# B&R Automation Studio project perfxxl (part 4)

#### xml_interface.c
```c
#ifdef _DEFAULT_INCLUDES
	#include <AsDefault.h>
#endif
/***************************************************************************/
/*                                                                         */
/* Datei:    xml_interface.c                                               */
/*                                                                         */
/* Autor:    Herbert Aden, Krause-Biagosch GmbH                            */
/*                                                                         */
/* Abstrakt: Diese Task wartet darauf, daß sich ein TCP-IP Client am ein-  */
/*           gestellten Port anmeldet.   Wenn die Verbindung hergestellt   */
/*           worden ist, schickt der server zyklisch XML codierte          */
/*           wird versucht, die Verbindung wieder neu aufzubauen.          */
/*                                                                         */
/* Datum:    08.12.2006       letzte Änderungen: 25.01.2007  / HA          */
/*                                                                         */
/***************************************************************************/

/***** Include-Files: *****/
#include <Ethernet.h>
#include <string.h>
#include <ctype.h>
#include <visapi.h>
#include "asstring.h"
#include "glob_var.h"
#include "EGMglob_var.h"

/***** Variablen-/Konstantendeklaration: *****/
/* Anwendungsspezifische Konstanten: */
#define TCP_IP_PORT		2020				/* Port für Kommunikation */
#define SEND_BUFFER_LEN	3000				/* Buffer-Länge für das Senden */
#define RECV_BUFFER_LEN	150					/* Empfangs-Buffer Länge */
#define TIMEOUT			200					/* Abbruch nach TIMEOUT * Zykluszeit Sek.*/
#define	RCVTIMEOUT		200
#define MAXCLIENTS		5
#define	LIVEBYTECNT		160
#define SEND_EVERY_N_SEC 5					/* send every 5 seconds an xml message*/

/* sonstige Konstanten */
#define TCP_IP_OK			0
#define TCP_IP_NO_RCV_DATA	27211
#define TCP_IP_BUSY		65535
#define TCPIPMGR_TIMEOUT 14893
#define BUF_ZERO 14896

#define OPEN_PORT			0
#define WAIT_OPEN_PORT		1
#define SEND_DATA			2
#define WAIT_SEND_DATA		3
#define RECV_DATA			4
#define WAIT_RECV_DATA		5
#define CLOSE_PORT			6
#define WAIT_CLOSE_PORT		7

#define MAXERRORS			51

/* Strukturen fuer Ethernet-Libraray-Funktionen */
_LOCAL    TCPserv_typ         TCP_Server[MAXCLIENTS];
_LOCAL    TCPrecv_typ         TCP_Recv[MAXCLIENTS];
_LOCAL    TCPsend_typ         TCP_Send[MAXCLIENTS];
_LOCAL    TCPclose_typ        TCP_Close[MAXCLIENTS];

_LOCAL    SINT                Step[MAXCLIENTS];
_LOCAL    UINT                RcvLength;
_LOCAL    USINT               Count[MAXCLIENTS];
_LOCAL    USINT               SendDataCnt[MAXCLIENTS];
/* Buffer for XML Message */
_LOCAL    SINT                XMLBuffer[SEND_BUFFER_LEN];
_LOCAL    UINT                SendTimeout[MAXCLIENTS];
_LOCAL    UINT                Len;
_LOCAL    UINT                DataLock;

/* Variablen: */
static    SINT                SendBuffer[MAXCLIENTS][SEND_BUFFER_LEN];
static    SINT                RecvBuffer[MAXCLIENTS][RECV_BUFFER_LEN];
static    SINT                RecvData[MAXCLIENTS][RECV_BUFFER_LEN];
static    BOOL                CloseConnection[MAXCLIENTS];
static    int                 CurrentClient,parse;
static    int                 i;

static const char *ErrorTexts[] =
{
	"Not-Aus",
	"kein Antriebstakt",
	"Gummierung Füllstand zu niedrig",
	"Vorspülen Füllstand zu niedrig",
	"Nachspülen Füllstand zu niedrig",
	"Entwickler Füllstand zu niedrig",
	"Entwickler Temperatur zu niedrig",
	"Entwickler Temperatur zu hoch",
	"Nacherwärmung 1 Temperatur zu niedrig",
	"Nacherwärmung 1 Temperatur zu hoch",
	"Nacherwärmung 2 Temperatur zu niedrig",
	"Nacherwärmung 2 Temperatur zu hoch",
	"Plattenstau",
	"Entwickler zu alt",
	"E/A Modul nicht gefunden",
	"Nacherwärmung Temperatur-Sensor 1 defekt",
	"Nacherwärmung Temperatur-Sensor 2 defekt",
	"Nacherwärmung Umgebungs-Sensor defekt",
	"Entwickler Temperatur-Sensor defekt",
	"Nacherwärmung Heizung 1 defekt",
	"Nacherwärmung Heizung 2 defekt",
	"Vorspülstation: Befüllen fehlgeschlagen",
	"Nachspülstation: Befüllen fehlgeschlagen",
	"Entwickler Befüllen fehlgeschlagen",
	"Nacherwärmung 1 überhitzt",
	"Nacherwärmung 2 überhitzt",
	"Entwickler überhitzt",
	"Antrieb Geschwindigkeitsabweichung zu groß",
	"Temperatur Modul nicht gefunden",
	"Digitales Eingangsmodul nicht gefunden",
	"Digitales Ausgangsmodul nicht gefunden",
	"Analoges Ausgangsmodul nicht gefunden",
	"Versorgungsmodul nicht gefunden",
	"Gummierung: Kein Durchfluß",
	"Entwicklerzirkulation: Kein Durchfluß",
	"Vorspülen: Kein Durchfluß",
	"Nachspülen: Kein Durchfluß",
	"Regenerat Kanister leer",
	"Entwickler Kanister leer",
	"Nacherw.: Heizung 3 defekt",
	"Nacherw.: Heizung 4 defekt",
	"Nacherwärmung Kreis 3 Temp. zu niedrig",
	"Nacherwärmung Kreis 3 Temp. zu hoch",
	"Nacherwärmung Kreis 4 Temp. zu niedrig",
	"Nacherwärmung Kreis 4 Temp. zu hoch",
	"Nacherwärmung Kreis 3 überhitzt",
	"Nacherwärmung Kreis 4 überhitzt",
	"Nacherw.: Temperaturfühler 3 defekt",
	"Nacherw.: Temperaturfühler 4 defekt",
	"Abwassertank fast voll!",
	"Abwassertank voll, Maschine gestoppt!",
	"EOL",	/* End of Errorlist (for detection in loop) */
	" ",
	" ",
	" ",
	" ",
	" ",
	" ",
	" "
};

/***** INIT FUNKTION *******************************************************/
_INIT void init (void)
{
	int i;
	CurrentClient = 1;
	/* Initialisierung der TCP-IP Datenstrukturen: */

	for(i = 0;i<MAXCLIENTS;i++)
	{
		SendDataCnt[i] = 0;
		/* TCP-IP Client: */
		TCP_Server[i].enable	= TRUE;
		TCP_Server[i].porta	= TCP_IP_PORT+i;

		/* TCP-IP Client Senden: */
		TCP_Send[i].enable		= TRUE;
		TCP_Send[i].buffer		= (UDINT)&SendBuffer[i][0];
		TCP_Send[i].buflng		= SEND_BUFFER_LEN;

		/* TCP-IP Client Empfangen: */
		TCP_Recv[i].enable		= TRUE;
		TCP_Recv[i].buffer		= (UDINT)&RecvBuffer[i][0];
		TCP_Recv[i].mxbuflng	= RECV_BUFFER_LEN;

		/* TCP-IP Client schließen */
		TCP_Close[i].enable	= TRUE;

		Step[i] = OPEN_PORT;
		Count[i] = 0;
		CloseConnection[i] = 0;
	}

} /* Ende Funktion _INIT void init (void) */

void CreateXMLMessage( USINT *buf)
{
	char tmp[20];
	char TempError[64];
	int i,ErrorNumber;

	void AddVal2(USINT *buf, char *before,char *Value, char *after)
	{
		strcat(buf,before);
		strcat(buf,Value);
		strcat(buf,after);
	}

	strcpy(buf,"<KrauseMessage>\r\n\t<Bluefin>\r\n\t\t<MachineName>Bluefin</MachineName>\r\n");

			strcat(buf,"\t\t<MachineNumber>");
			strncat(buf,EGMGlobalParam.MachineNumber,9);
			strcat(buf,"</MachineNumber>\r\n");

			strcat(buf,"\t\t<MachineState>\r\n\t\t\t<State>");
/* Status Message*/
				strcpy(TempError,"No error");
				ErrorNumber = 0;
				switch (EGMState.mode)
				{
					case (M_OFF):
					case (M_CLEANING):
					case (M_INITCLEANING):
					{
					    if( !(ControlVoltageOk &&  ActivateControlVoltage) )
							strcat(buf,"EMERGENCY</State>\r\n\t\t\t<ErrorNumber>");
						else
							strcat(buf,"STANDBY</State>\r\n\t\t\t<ErrorNumber>");
						break;
					}
					case (M_AUTO):
					{
						switch (EGMState.state)
						{
							case (S_READY):
							{
								strcat(buf,"READY</State>\r\n\t\t\t<ErrorNumber>");
								break;
							}
							case (S_OFF):
							case (S_HEATING):
							{
								strcat(buf,"STANDBY</State>\r\n\t\t\t<ErrorNumber>");
								break;
							}
							case (S_STARTPROCESSING):
							case (S_PROCESSING):
							case (S_WAITFORSTANDBY):
							{
								strcat(buf,"BUSY</State>\r\n\t\t\t<ErrorNumber>");
								break;
							}
							case (S_ERROR):
							{
								BOOL Err = FALSE;
								strcat(buf,"ERROR</State>\r\n\t\t\t<ErrorNumber>");
/* find 1st error in list */
								for(i=0;i<MAXERRORS;i++)
								{
									if (EGM_AlarmBitField[i] == TRUE)
										break;
/* safety: detect End of Errorlist */
									if( strcmp(ErrorTexts[i],"EOL") == 0 )
									{
										Err = TRUE;
										break;
									}

								}
/* safety: End of Errorlist was detected */
								if(!Err && i<MAXERRORS)
								{
									strncpy(TempError,ErrorTexts[i],sizeof(TempError)-1);
									ErrorNumber = i;
								}
								else
								{
									ErrorNumber = 0;
								}
								break;
							}
						}
						break;
					}

				}
				itoa(ErrorNumber,(UDINT )&tmp[0]);
				strcat(buf,tmp);
				strcat(buf,"</ErrorNumber>\r\n\t\t\t<ErrorDescription>");
				strcat(buf,TempError);
				strcat(buf,"</ErrorDescription>\r\n\t\t\t<Errorlist>");
				for(i=0;i<EGM_MAXALARMS;i++)
				{
					if(EGM_AlarmBitField[i])
						strcat(buf,"1");
					else
						strcat(buf,"0");
				}

				strcat(buf,"</Errorlist>\r\n\t\t\t<StateCode>");
/* Emergency stop soll auch zu Error führen:*/
			    if( !(ControlVoltageOk &&  ActivateControlVoltage) )
					itoa(S_ERROR,(UDINT )&tmp[0]);
			    else
					itoa(EGMState.state,(UDINT )&tmp[0]);
				strcat(buf,tmp);
				strcat(buf,"</StateCode>\r\n\t\t</MachineState>\r\n\t\t<MachineParam>\r\n\t\t\t<PreHeat>\r\n");
/* Preheat values*/
					ftoa((REAL)EGMPreheat.RealTemp[0]/10.0,(UDINT )&tmp[0]);
					AddVal2(buf, "\t\t\t\t<Temperature1>\r\n\t\t\t\t\t<Description>Heating 1</Description>\r\n\t\t\t\t\t<Type>double</Type>\r\n\t\t\t\t\t<Value>", tmp,
					"</Value>\r\n\t\t\t\t\t<Unit>deg. C</Unit>\r\n\t\t\t\t</Temperature1>\r\n");
					ftoa((REAL)EGMPreheat.RealTemp[1]/10.0,(UDINT )&tmp[0]);
					AddVal2(buf, "\t\t\t\t<Temperature2>\r\n\t\t\t\t\t<Description>Heating 2</Description>\r\n\t\t\t\t\t<Type>double</Type>\r\n\t\t\t\t\t<Value>", tmp,
					"</Value>\r\n\t\t\t\t\t<Unit>deg. C</Unit>\r\n\t\t\t\t</Temperature2>\r\n");
					ftoa((REAL)EGMPreheat.RealTemp[2]/10.0,(UDINT )&tmp[0]);
					AddVal2(buf, "\t\t\t\t<Temperature3>\r\n\t\t\t\t\t<Description>Ambient</Description>\r\n\t\t\t\t\t<Type>double</Type>\r\n\t\t\t\t\t<Value>", tmp,
					"</Value>\r\n\t\t\t\t\t<Unit>deg. C</Unit>\r\n\t\t\t\t</Temperature3>\r\n\t\t\t</PreHeat>\r\n\t\t\t<Developer>\r\n");
/* Developer values */
					ftoa((REAL)EGMDeveloperTank.RealTemp/10.0,(UDINT )&tmp[0]);
					AddVal2(buf, "\t\t\t\t<Temperature1>\r\n\t\t\t\t\t<Description>Temperature of fluid</Description>\r\n\t\t\t\t\t<Type>double</Type>\r\n\t\t\t\t\t<Value>", tmp,
					"</Value>\r\n\t\t\t\t\t<Unit>deg. C</Unit>\r\n\t\t\t\t</Temperature1>\r\n");
					if(EGMDeveloperTank.LevelInRange)
						strcat(buf,"\t\t\t\t<LevelOK>\r\n\t\t\t\t\t<Description>Level of developer</Description>\r\n\t\t\t\t\t<Type>boolean</Type>\r\n\t\t\t\t\t<Value>true</Value>\r\n\t\t\t\t</LevelOK>\r\n\t\t\t</Developer>\r\n\t\t\t<Speeds>\r\n");
					else
						strcat(buf,"\t\t\t\t<LevelOK>\r\n\t\t\t\t\t<Description>Level of developer</Description>\r\n\t\t\t\t\t<Type>boolean</Type>\r\n\t\t\t\t\t<Value>false</Value>\r\n\t\t\t\t</LevelOK>\r\n\t\t\t</Developer>\r\n\t\t\t<Speeds>\r\n");
					ftoa(EGMGlobalParam.CurrentPlateSpeed,(UDINT )&tmp[0]);
					AddVal2(buf, "\t\t\t\t<PlateSpeedAct>\r\n\t\t\t\t\t<Description>Actual speed (measured)</Description>\r\n\t\t\t\t\t<Type>double</Type>\r\n\t\t\t\t\t<Value>", tmp,
					"</Value>\r\n\t\t\t\t\t<Unit>m per min</Unit>\r\n\t\t\t\t</PlateSpeedAct>\r\n");
					ftoa((EGMGlobalParam.MainMotorFactor*EGMMainMotor.RatedRpm),(UDINT )&tmp[0]);
					AddVal2(buf, "\t\t\t\t<PlateSpeedRef>\r\n\t\t\t\t\t<Description>Referenced speed</Description>\r\n\t\t\t\t\t<Type>double</Type>\r\n\t\t\t\t\t<Value>", tmp,
					"</Value>\r\n\t\t\t\t\t<Unit>m per min</Unit>\r\n\t\t\t\t</PlateSpeedRef>\r\n");
					itoa(EGMBrushMotor.RatedRpm*EGMGlobalParam.BrushFactor,(UDINT )&tmp[0]);
					AddVal2(buf, "\t\t\t\t<BrushSpeed>\r\n\t\t\t\t\t<Description>Speed of brushes</Description>\r\n\t\t\t\t\t<Type>int</Type>\r\n\t\t\t\t\t<Value>", tmp,
/*					"</Value>\r\n\t\t\t\t\t<Unit>rpm</Unit>\r\n\t\t\t\t</BrushSpeed>\r\n\t\t\t</Speeds>\r\n\t\t</MachineParam>\r\n\t</Bluefin>\r\n</KrauseMessage>\r\n");*/
/* *** */
					"</Value>\r\n\t\t\t\t\t<Unit>rpm</Unit>\r\n\t\t\t\t</BrushSpeed>\r\n\t\t\t</Speeds>\r\n\t\t</MachineParam>\r\n");
/* Verbrauchsdaten */
				strcat(buf,"\t\t<PlateCountValues>\r\n");
					itoa(OverallPlateCounter,(UDINT )&tmp[0]);
					AddVal2(buf, "\t\t\t<OverallPlates>\r\n\t\t\t\t<Description>Plates processed (overall)</Description>\r\n\t\t\t\t<Type>int</Type>\r\n\t\t\t\t<Value>", tmp,
					"</Value>\r\n\t\t\t\t<Unit>pcs.</Unit>\r\n\t\t\t</OverallPlates>\r\n");
					itoa(SessionPlateCounter,(UDINT )&tmp[0]);
					AddVal2(buf, "\t\t\t<SessionPlates>\r\n\t\t\t\t<Description>Plates processed since power on</Description>\r\n\t\t\t\t<Type>int</Type>\r\n\t\t\t\t<Value>", tmp,
					"</Value>\r\n\t\t\t\t<Unit>pcs.</Unit>\r\n\t\t\t</SessionPlates>\r\n");
					ftoa(OverallSqmCounter,(UDINT )&tmp[0]);
					AddVal2(buf, "\t\t\t<OverallSqm>\r\n\t\t\t\t<Description>Squaremeters processed (overall)</Description>\r\n\t\t\t\t<Type>double</Type>\r\n\t\t\t\t<Value>", tmp,
					"</Value>\r\n\t\t\t\t<Unit>sqm</Unit>\r\n\t\t\t</OverallSqm>\r\n");
					ftoa(SessionSqmCounter,(UDINT )&tmp[0]);
					AddVal2(buf, "\t\t\t<SessionSqm>\r\n\t\t\t\t<Description>Squaremeters processed since power on</Description>\r\n\t\t\t\t<Type>double</Type>\r\n\t\t\t\t<Value>", tmp,
					"</Value>\r\n\t\t\t\t<Unit>sqm</Unit>\r\n\t\t\t</SessionSqm>\r\n\t\t</PlateCountValues>\r\n");
/* Version */
				strcat(buf,"\t\t<Version>");
				strcat(buf,gVERSION);
				strcat(buf,"</Version>\r\n\t</Bluefin>\r\n</KrauseMessage>\r\n");

/* safety */
	if(strlen(buf) > SEND_BUFFER_LEN)
		buf[SEND_BUFFER_LEN-1] = 0;
	return;
}

/***** ZYKLISCHE FUNKTION **************************************************/
_CYCLIC void cyclic (void)
{

	if ( DataLock == 0 )
		CreateXMLMessage( (USINT *)&XMLBuffer[0] );

	for(CurrentClient = 0;CurrentClient<MAXCLIENTS;CurrentClient++)
	{
	/***** Öffnen des Ports ************************************************/
		if (Step[CurrentClient] == OPEN_PORT)
		{
 			CloseConnection[CurrentClient] = 0;
			/* 1. Aufruf der Funktion */
			TCPserv (&TCP_Server[CurrentClient]);
			/* Status prüfen: */
			if (TCP_Server[CurrentClient].status == TCP_IP_OK)
			{
				/* Port geöffnet */
				/* Identifier zuordnen ... */
				TCP_Send[CurrentClient].cident = TCP_Server[CurrentClient].cident;
				TCP_Recv[CurrentClient].cident = TCP_Server[CurrentClient].cident;
				TCP_Close[CurrentClient].cident = TCP_Server[CurrentClient].cident;
				/* ... und zum nächsten Schritt gehen */
				Step[CurrentClient] = RECV_DATA;
				SendTimeout[CurrentClient] = 0;
			}
		} /* if (Step == WAIT_OPEN_PORT) */

	/***** Daten Empfangen *************************************************/
		if (Step[CurrentClient] == RECV_DATA)
		{
			TCPrecv (&TCP_Recv[CurrentClient]);
			/* Status prüfen: */
			if (TCP_Recv[CurrentClient].status == TCP_IP_OK)
			{
				if(TCP_Recv[CurrentClient].rxbuflng == 0) /*CLOSE von Gegenstelle*/
				{
					Step[CurrentClient] = CLOSE_PORT;
					Count[CurrentClient] = 0;
				}
				else	/* Daten empfangen -> auswerten*/
				{
					parse = 0;
					/*einzelne Zeichen (via telnet)*/
					if(TCP_Recv[CurrentClient].rxbuflng < 3)
					{
						RecvData[CurrentClient][Count[CurrentClient]] = RecvBuffer[CurrentClient][0];
						Count[CurrentClient]++;
/* safety !*/
						if (Count[CurrentClient] >= RECV_BUFFER_LEN )
						{
							strcpy(SendBuffer[CurrentClient],"HEY! \a\aSTOP SENDING!!");
							Step[CurrentClient] = SEND_DATA;
							TCP_Send[CurrentClient].buffer		= (UDINT)&SendBuffer[CurrentClient];
							TCP_Send[CurrentClient].buflng = strlen(SendBuffer[CurrentClient]);
							Count[CurrentClient] = 0;
							parse = 0;
						}
						else
						if( RecvBuffer[CurrentClient][0] == 10 || RecvBuffer[CurrentClient][0] == 13 )
						{
							RecvData[CurrentClient][Count[CurrentClient]] = 0;
							parse = 1;
						}
					}
					else
					{
						memcpy(RecvData[CurrentClient],RecvBuffer[CurrentClient],TCP_Recv[CurrentClient].rxbuflng);
						Count[CurrentClient] = TCP_Recv[CurrentClient].rxbuflng;
						parse = 1;
					}

					if(parse)
					{
						i=0;
						while(  ( RecvData[CurrentClient][i] != 0 )
						     && ( i < RECV_BUFFER_LEN) )
						{
							RecvData[CurrentClient][i] = toupper( RecvData[CurrentClient][i] );
							i++;
						}
						RecvData[CurrentClient][Count[CurrentClient]-1] = 0;

						if (strncmp(RecvData[CurrentClient],"BYE",3) == 0
						||	strncmp(RecvData[CurrentClient],"QUIT",4) == 0
						||	strncmp(RecvData[CurrentClient],"EXIT",4) == 0)
						{
							strcpy(SendBuffer[CurrentClient],"Good bye, cu next time...\r\n");
							CloseConnection[CurrentClient] = 1;
						}
						Step[CurrentClient] = SEND_DATA;
						TCP_Send[CurrentClient].buffer		= (UDINT)&SendBuffer[CurrentClient];
						TCP_Send[CurrentClient].buflng = strlen(SendBuffer[CurrentClient]);
						Count[CurrentClient] = 0;
						parse = 0;
					}
					SendDataCnt[CurrentClient]=0;
				}
			}
			else
			{
/*nothing received: ok, send from time to time*/
				SendDataCnt[CurrentClient]++;
				if( SendDataCnt[CurrentClient] >= 10*SEND_EVERY_N_SEC)
				{
					memcpy(SendBuffer[CurrentClient],XMLBuffer,sizeof(XMLBuffer));
					TCP_Send[CurrentClient].buflng = strlen(SendBuffer[CurrentClient]);
					Step[CurrentClient] = SEND_DATA;
					SendDataCnt[CurrentClient] = 0;
				}
			}
		}

/************** senden ****************************/

		if (Step[CurrentClient] == SEND_DATA)
		{

			TCPsend (&TCP_Send[CurrentClient]);
			/* Status prüfen: */
			if (TCP_Send[CurrentClient].status == TCP_IP_OK)
			{
				/* Senden war OK */
				if (CloseConnection[CurrentClient])
					Step[CurrentClient] = CLOSE_PORT;
				else
					Step[CurrentClient] = RECV_DATA;
				CloseConnection[CurrentClient] = 0;
				SendTimeout[CurrentClient] = 0;
			}
			else
			if (TCP_Send[CurrentClient].status == TCP_IP_BUSY)
			{
			/* VOID, just wait*/
			}
			else
			if (TCP_Send[CurrentClient].status == ERR_ETH_NET_SLOW)
			{
			/* Check for timeout, after 3 sec close the port and wait for reconnection */
				SendTimeout[CurrentClient]++;
				if(SendTimeout[CurrentClient] > 30) /* 3 sec*/
					Step[CurrentClient] = CLOSE_PORT;
			}
			else
			if (TCP_Send[CurrentClient].status == TCPIPMGR_TIMEOUT)
			{
			/* VOID, just wait*/
			}
			else	/* any other state, close after a certain time*/
			{
				SendTimeout[CurrentClient]++;
				if(SendTimeout[CurrentClient] > 30) /* 3 sec*/
					Step[CurrentClient] = CLOSE_PORT;
			}
		}

	/***** Port schließen **************************************************/
		if (Step[CurrentClient] == CLOSE_PORT)
		{
			SendTimeout[CurrentClient] = 0;
			TCPclose (&TCP_Close[CurrentClient]);
			/* Status prüfen: */
			if (TCP_Close[CurrentClient].status == TCP_IP_OK)
			{
				/* Port geschlossen, neu öffnen: */
				Step[CurrentClient] = OPEN_PORT;
			}
		} /* if (Step == WAIT_CLOSE_PORT) */

	} /*for*/

} /* Ende Funktion _CYCLIC void cyclic (void) */

/* ENDE */
```

### Program Logical/bluefin (ANSIC, version 0.00.0)

#### ifbluefin.c
```c
#ifdef _DEFAULT_INCLUDES
	#include <AsDefault.h>
#endif
/*
                             *******************
******************************* C SOURCE FILE *******************************
**                           *******************                           **
**                                                                         **
** project  : LS JET II                                                    **
** filename : IFBLUEFIN.C                                                  **
** version  : 1.01                                                         **
** date     : 23.06.2010                                                   **
**                                                                         **
*****************************************************************************
** Abstract                                                                **
** ========                                                                **
** -Interface to Bluefin via CAN using the IMA library                     **
**  Needs Dataobject DO_IMA                                                **
** -TCPIP Server for data transfer to BluefinServer, takes messages        **
**  from Bluefin (in connected XMLBuffer array) and transfers this         **
**  to all connected clients (max 3) periodically                          **
**  if no connection to Bluefin is established the message "BLUEFIN OFF"   **
**  is sent periodically                                                   **
**                                                                         **
** Copyright (c) 2006, Krause-Biagosch GmbH                                **
** All rights reserved.                                                    **
**                                                                         **
*****************************************************************************
VERSION HISTORY:
----------------
Version     : 1.00
Date        : 15.01.2007
Revised by  : Herbert Aden
Description : Original version.

Version     : 1.01
Date        : 23.06.2010
Revised by  : Herbert Aden
Description : Improved version from LSJet.

*/
#define _IFBLUEFIN_C_SRC

/****************************************************************************/
/**                                                                        **/
/**                           INCLUDE FILES                                **/
/**                                                                        **/
/****************************************************************************/
#include "glob_var.h"
#include "egmglob_var.h"
#include "in_out.h"
#include <AsIMA.h>
#include <Ethernet.h>
#include <string.h>
#include <ctype.h>
#include "asstring.h"

/****************************************************************************/
/**                                                                        **/
/**                       DEFINITIONS AND MACROS                           **/
/**                                                                        **/
/****************************************************************************/
#define IMA_CONN_OK          (0)

#define TCP_IP_PORT		2020				/* Port für Kommunikation */
#define SEND_BUFFER_LEN	3000				/* Buffer-Länge für das Senden */
#define OLD_SEND_BUFFER_LEN	2500				/* XML Buffer-Länge für Bluefin <=2.10*/
#define RECV_BUFFER_LEN	150					/* Empfangs-Buffer Länge */
#define TIMEOUT			200					/* Abbruch nach TIMEOUT * Zykluszeit Sek.*/
#define	RCVTIMEOUT		200
#define MAXCLIENTS		3
#define	LIVEBYTECNT		160
#define SEND_EVERY_N_SEC 3					/* send every 5 seconds an xml message*/

/* sonstige Konstanten */
#define TCP_IP_OK			0
#define TCP_IP_NO_RCV_DATA	27211
#define TCP_IP_BUSY		65535
#define TCPIPMGR_TIMEOUT 14893
#define BUF_ZERO 14896

#define OPEN_PORT			0
#define WAIT_OPEN_PORT		1
#define SEND_DATA			2
#define WAIT_SEND_DATA		3
#define RECV_DATA			4
#define WAIT_RECV_DATA		5
#define CLOSE_PORT			6
#define WAIT_CLOSE_PORT		7
#define WAIT				8
#define PREPARE_SEND_DATA   9

/****************************************************************************/
/**                                                                        **/
/**                      TYPEDEFS AND STRUCTURES                           **/
/**                                                                        **/
/****************************************************************************/
/* NONE */

/****************************************************************************/
/**                                                                        **/
/**                      PROTOTYPES OF LOCAL FUNCTIONS                     **/
/**                                                                        **/
/****************************************************************************/
/* NONE */

/****************************************************************************/
/**                                                                        **/
/**                      EXPORTED VARIABLES                                **/
/**                                                                        **/
/****************************************************************************/
/* NONE */

/****************************************************************************/
/**                                                                        **/
/**                           GLOBAL VARIABLES                             **/
/**                                                                        **/
/****************************************************************************/

/****************************************************************************/
/**                                                                        **/
/**                      TASK-LOCAL VARIABLES                              **/
/**                                                                        **/
/****************************************************************************/
_LOCAL    INT                 IMAStatusInit,IMAStatusComm;
_LOCAL    imaInfoStruct       errorInfo,ConnInfoPV,ConnInfoAUX;
_LOCAL    UDINT               IMAident;

_LOCAL    INT                 IMAStatusInitVCP,IMAStatusInitXSOld,IMAStatusCommVCP,IMAStatusCommXSOld;
_LOCAL    imaInfoStruct       errorInfoVCP,ConnInfoPVVCP,ConnInfoAUXVCP;
_LOCAL    imaInfoStruct       errorInfoXSOld,ConnInfoPVXSOld,ConnInfoAUXXSOld;
_LOCAL    UDINT               IMAidentVCP,IMAidentXSOld;

_LOCAL    UINT                byte_link_cnt;

/* structs for Ethernet-Library-Functions */
_LOCAL	TCPserv_typ			TCP_Server[MAXCLIENTS];
_LOCAL	TCPrecv_typ			TCP_Recv[MAXCLIENTS];
_LOCAL	TCPsend_typ			TCP_Send[MAXCLIENTS];
_LOCAL	TCPclose_typ		TCP_Close[MAXCLIENTS];
_LOCAL	SINT	Step[MAXCLIENTS];
_LOCAL	UINT	SendTimeout[MAXCLIENTS];
_LOCAL	UINT	RcvLength;

/* Buffer for XML Message */
_LOCAL SINT	XMLBuffer[SEND_BUFFER_LEN];
_LOCAL SINT	OldXMLBuffer[OLD_SEND_BUFFER_LEN];
_LOCAL UINT EnablePVComm;
_LOCAL UINT	DataLock;
_LOCAL BOOL                CAN_EGM1;
_LOCAL BOOL                CAN_EGM2;
_LOCAL BOOL                CAN_VCP;
_LOCAL STRING              BFVERSION[9];
_LOCAL UINT                IMACommStep;
_LOCAL UINT                VisConnOK;

/****************************************************************************/
/**                                                                        **/
/**                    MODULE-LOCAL VARIABLES                              **/
/**                                                                        **/
/****************************************************************************/
/* for IMA Comm */
static    STRING              DOName[32]="do_ima";
static    STRING              DONameVCP[32]="do_vcp";
static    STRING              DONameXSOld[32]="do_xsold";
/* for Ethernet server */
static    SINT                SendBuffer[MAXCLIENTS][SEND_BUFFER_LEN];
static    SINT                RecvBuffer[MAXCLIENTS][RECV_BUFFER_LEN];
static    SINT                RecvData[MAXCLIENTS][RECV_BUFFER_LEN];

static    int                 CurrentClient,parse;
static    USINT               Count[MAXCLIENTS];
static    int                 i;
static    USINT               SendDataCnt[MAXCLIENTS];
static    BOOL                CloseConnection[MAXCLIENTS];
static    UINT                NumberOfFreePorts;
static    UINT                WaitCounter[MAXCLIENTS];
static    BOOL                ConnectedTo3000Byte;
/****************************************************************************/
/**                                                                        **/
/**                          LOCAL FUNCTIONS                               **/
/**                                                                        **/
/****************************************************************************/
_INIT void InitFunc(void)
{
#ifdef MODE_PERFORMANCE
	int i;
	ConnectedTo3000Byte = FALSE;
	IMACommStep = 0;
	IMAStatusInit = IMAinit((UDINT)DOName, &errorInfo, &IMAident);
	IMAStatusInitVCP = IMAinit((UDINT)DONameVCP, &errorInfoVCP, &IMAidentVCP);
	IMAStatusInitXSOld = IMAinit((UDINT)DONameXSOld, &errorInfoXSOld, &IMAidentXSOld);

	CurrentClient = 1;
	/* Initialise TCP-IP Data structs: */
	for(i = 0;i<MAXCLIENTS;i++)
	{
		SendDataCnt[i] = 0;
		/* TCP-IP Client: */
		TCP_Server[i].enable	= TRUE;
		TCP_Server[i].porta	= TCP_IP_PORT+i;

		/* TCP-IP Client Senden: */
		TCP_Send[i].enable		= TRUE;
		TCP_Send[i].buffer		= (UDINT)&SendBuffer[i][0];
		TCP_Send[i].buflng		= SEND_BUFFER_LEN;

		/* TCP-IP Client Empfangen: */
		TCP_Recv[i].enable		= TRUE;
		TCP_Recv[i].buffer		= (UDINT)&RecvBuffer[i][0];
		TCP_Recv[i].mxbuflng	= RECV_BUFFER_LEN;

		/* TCP-IP Client schließen */
		TCP_Close[i].enable	= TRUE;

		Step[i] = OPEN_PORT;
		Count[i] = 0;
		CloseConnection[i] = 0;
	}
	NumberOfFreePorts = MAXCLIENTS;
	AlarmBitField[35] = FALSE;
	VisConnOK = 0;
#endif
}

_CYCLIC void CyclicFunc(void)
{
/*****************************************************************************/
/* get data from Bluefin via INA comm */
/*****************************************************************************/

#ifdef MODE_BOTH
/* Performance und Bluefin: EGM Signale direkt aus der Software*/
	StatusEGM1 = NoError;
	StatusEGM2 = Ready;
	VCP = VCP_OK;
#else
/* Performance allein: EGM Signale via CAN Anbindung oder Eingänge*/

	if(IMAStatusInit == IMA_OK)  /* Init was OK (should always be the case) */
	{
		switch (IMACommStep)
		{
			case 0:
			{ /* Versuch, mit der neuesten Version zu connecten */
				IMAStatusCommVCP = IMAcomm(IMAidentVCP, &ConnInfoPVVCP, &ConnInfoAUXVCP);

				if(IMAStatusCommVCP == IMA_OK)
				{
/*
 * Bluefin XS Version bis 3.04 hat 2500 Byte Puffer, deswegen dann anderen
 * Verbindungs DB benutzen
 */
					if(  (BFVERSION[0] == '3')
					  && (BFVERSION[2] == '0')
					  && (BFVERSION[5] != 'L') /* LC Version erkennen, die hat nämlich
					                            * auch 3000 Byte und VCP Verbindung
					                            */
				  )
					{
						IMACommStep = 20;
					}
					else
					{
						ConnectedTo3000Byte = TRUE;
						StatusEGM1 = CAN_EGM1;
						StatusEGM2 = CAN_EGM2;
						VCP = CAN_VCP;
						AlarmBitField[35] = FALSE;
						VisConnOK = 1;

						if(NumberOfFreePorts < MAXCLIENTS)
							EnablePVComm = 1;
						else
							EnablePVComm = 0;
					}
				}
				else /* fehlgeschlagen: Verbindung beenden und alte Version probieren */
					IMACommStep = 20;
				break;
			}

			case 20:
			{ /* Versuch, mit Version XS mit 2500 Byte zu connecten */
				IMAStatusCommXSOld = IMAcomm(IMAidentXSOld, &ConnInfoPVXSOld, &ConnInfoAUXXSOld);

				if(IMAStatusCommXSOld == IMA_OK)
				{
					ConnectedTo3000Byte = FALSE;
					StatusEGM1 = CAN_EGM1;
					StatusEGM2 = CAN_EGM2;
					VCP = CAN_VCP;
					AlarmBitField[35] = FALSE;
					VisConnOK = 1;

					if(NumberOfFreePorts < MAXCLIENTS)
						EnablePVComm = 1;
					else
						EnablePVComm = 0;
				}
				else /* fehlgeschlagen: Verbindung beenden und alte Version probieren */
					IMACommStep = 30;
				break;
			}

			case 30:
			{ /* Versuch, mit der alten Version zu connecten */
				IMAStatusComm = IMAcomm(IMAident, &ConnInfoPV, &ConnInfoAUX);

				if(IMAStatusComm == IMA_OK)
				{
/*
 * Bluefin XS Version bis 3.04 hat auch 2500 Byte Puffer, wird nicht per Fehler erkannt,
 * weil hier (im hierzu gehörigen DB) nicht auf CAN_VCP zugegriffen wird
 * deshalb über Versionsnummer
 */
					if(  (BFVERSION[0] == '3')
					  )
					{
						IMACommStep = 20;
					}
					else
					{
						ConnectedTo3000Byte = FALSE;
						StatusEGM1 = CAN_EGM1;
						StatusEGM2 = CAN_EGM2;
						VCP = CAN_VCP;
						AlarmBitField[35] = FALSE;
						VisConnOK = 1;

						if(NumberOfFreePorts < MAXCLIENTS)
							EnablePVComm = 1;
						else
							EnablePVComm = 0;
					}
				}
				else /* fehlgeschlagen: Fehlermeldung und von vorn beginnen */
				{
					ConnInfoPVVCP.commandClearError = TRUE;
					ConnInfoPVXSOld.commandClearError = TRUE;
					ConnInfoPV.commandClearError = TRUE;
					VisConnOK = 0;
					IMACommStep = 0;
					StatusEGM1 = InEGM1;
					StatusEGM2 = InEGM2;
					VCP = In_VCPOK;
					break;
				}
				break;
			}
		}/*switch*/
	}
	else  /* comm not OK: EGM signals via Digital inputs*/
	{
		ConnectedTo3000Byte = FALSE;
		StatusEGM1 = InEGM1;
		StatusEGM2 = InEGM2;
		VCP = In_VCPOK;
	}

/*****************************************************************************/
/* TCP/IP Server */
/*****************************************************************************/
	NumberOfFreePorts = 0;

	for(CurrentClient = 0;CurrentClient<MAXCLIENTS;CurrentClient++)
	{
	/***** Öffnen des Ports ************************************************/
		if (Step[CurrentClient] == OPEN_PORT)
		{
 			CloseConnection[CurrentClient] = 0;
			/* 1. Aufruf der Funktion */
			TCPserv (&TCP_Server[CurrentClient]);
			/* Status prüfen: */
			if (TCP_Server[CurrentClient].status == TCP_IP_OK)
			{
				/* Port geöffnet */
				/* Identifier zuordnen ... */
				TCP_Send[CurrentClient].cident = TCP_Server[CurrentClient].cident;
				TCP_Recv[CurrentClient].cident = TCP_Server[CurrentClient].cident;
				TCP_Close[CurrentClient].cident = TCP_Server[CurrentClient].cident;
				/* ... und zum nächsten Schritt gehen */
				Step[CurrentClient] = RECV_DATA;
				SendTimeout[CurrentClient] = 0;
			}
			else
				NumberOfFreePorts++;
		} /* if (Step == WAIT_OPEN_PORT) */

	/***** Daten Empfangen *************************************************/
		if (Step[CurrentClient] == RECV_DATA)
		{
			TCPrecv (&TCP_Recv[CurrentClient]);
			/* Status prüfen: */
			if (TCP_Recv[CurrentClient].status == TCP_IP_OK)
			{
				if(TCP_Recv[CurrentClient].rxbuflng == 0) /*CLOSE von Gegenstelle*/
				{
					Step[CurrentClient] = CLOSE_PORT;
					Count[CurrentClient] = 0;
				}
				else	/* Daten empfangen -> auswerten*/
				{
					parse = 0;
					/*einzelne Zeichen (via telnet)*/
					if(TCP_Recv[CurrentClient].rxbuflng < 3)
					{
						RecvData[CurrentClient][Count[CurrentClient]] = RecvBuffer[CurrentClient][0];
						Count[CurrentClient]++;
/* safety !*/
						if (Count[CurrentClient] >= RECV_BUFFER_LEN )
						{
							strcpy(SendBuffer[CurrentClient],"HEY! \a\aSTOP SENDING!!");
							Step[CurrentClient] = SEND_DATA;
							TCP_Send[CurrentClient].buffer		= (UDINT)&SendBuffer[CurrentClient];
							TCP_Send[CurrentClient].buflng = strlen(SendBuffer[CurrentClient]);
							Count[CurrentClient] = 0;
							parse = 0;
						}
						else
						if( RecvBuffer[CurrentClient][0] == 10 || RecvBuffer[CurrentClient][0] == 13 )
						{
							RecvData[CurrentClient][Count[CurrentClient]] = 0;
							parse = 1;
						}
					}
					else
					{
						memcpy(RecvData[CurrentClient],RecvBuffer[CurrentClient],TCP_Recv[CurrentClient].rxbuflng);
						Count[CurrentClient] = TCP_Recv[CurrentClient].rxbuflng;
						parse = 1;
					}

					if(parse)
					{
						i=0;
						while(  ( RecvData[CurrentClient][i] != 0 )
						     && ( i < RECV_BUFFER_LEN) )
						{
							RecvData[CurrentClient][i] = toupper( RecvData[CurrentClient][i] );
							i++;
						}
						RecvData[CurrentClient][Count[CurrentClient]-1] = 0;

						if (strncmp(RecvData[CurrentClient],"BYE",3) == 0
						||	strncmp(RecvData[CurrentClient],"QUIT",4) == 0
						||	strncmp(RecvData[CurrentClient],"EXIT",4) == 0)
						{
							strcpy(SendBuffer[CurrentClient],"Good bye, cu next time...\r\n");
							CloseConnection[CurrentClient] = 1;
						}
						Step[CurrentClient] = SEND_DATA;
						TCP_Send[CurrentClient].buffer		= (UDINT)&SendBuffer[CurrentClient];
						TCP_Send[CurrentClient].buflng = strlen(SendBuffer[CurrentClient]);
						Count[CurrentClient] = 0;
						parse = 0;
					}
					SendDataCnt[CurrentClient]=0;
				}
			}
			else
			{
/*nothing received: ok, send from time to time*/
				SendDataCnt[CurrentClient]++;
				if( SendDataCnt[CurrentClient] >= 10*SEND_EVERY_N_SEC )
				{
					if(  (IMAStatusComm    == IMA_OK)
					 ||  (IMAStatusCommVCP == IMA_OK)
					 ||  (IMAStatusCommXSOld == IMA_OK) )
					{
						DataLock = 1;
						Step[CurrentClient] = WAIT;
						SendDataCnt[CurrentClient] = 0;
						WaitCounter[CurrentClient] = 0;
					}
					else
					{
						strcpy(SendBuffer[CurrentClient],"BLUEFIN OFF");
						TCP_Send[CurrentClient].buflng = strlen(SendBuffer[CurrentClient]);
						Step[CurrentClient] = SEND_DATA;
						SendDataCnt[CurrentClient] = 0;
					}
				}
			}
		}

/* SENDEDATEN VORBEREITEN */
		if (Step[CurrentClient] == PREPARE_SEND_DATA)
		{
			if(ConnectedTo3000Byte)
			{
/* Bluefin XS Version mit 3000 Byte xml Puffer */
				if( strncmp(XMLBuffer,"<KrauseMessage>",15) == 0 )
				{
					memcpy(SendBuffer[CurrentClient],XMLBuffer,sizeof(XMLBuffer));
					TCP_Send[CurrentClient].buflng = strlen(SendBuffer[CurrentClient]);
					Step[CurrentClient] = SEND_DATA;
					SendDataCnt[CurrentClient] = 0;
					DataLock = 0;
				}
			}
			else
			{
/* Bluefin standard Version mit 2500 Byte xml Puffer */
				if( strncmp(OldXMLBuffer,"<KrauseMessage>",15) == 0 )
				{
					memcpy(SendBuffer[CurrentClient],OldXMLBuffer,sizeof(OldXMLBuffer));
					SendBuffer[CurrentClient][sizeof(OldXMLBuffer)-1] = 0;
					TCP_Send[CurrentClient].buflng = strlen(SendBuffer[CurrentClient]);
					Step[CurrentClient] = SEND_DATA;
					SendDataCnt[CurrentClient] = 0;
					DataLock = 0;
				}
			}
		}

/************** senden ****************************/

		if (Step[CurrentClient] == SEND_DATA)
		{

			TCPsend (&TCP_Send[CurrentClient]);
			/* Status prüfen: */
			if (TCP_Send[CurrentClient].status == TCP_IP_OK)
			{
				/* Senden war OK */
				if (CloseConnection[CurrentClient])
					Step[CurrentClient] = CLOSE_PORT;
				else
					Step[CurrentClient] = RECV_DATA;
				CloseConnection[CurrentClient] = 0;
				SendTimeout[CurrentClient] = 0;
			}
			else
			if (TCP_Send[CurrentClient].status == TCP_IP_BUSY)
			{
			/* VOID, just wait*/
			}
			else
			if (TCP_Send[CurrentClient].status == ERR_ETH_NET_SLOW)
			{
			/* Check for timeout, after 3 sec close the port and wait for reconnection */
				SendTimeout[CurrentClient]++;
				if(SendTimeout[CurrentClient] > 30) /* 3 sec*/
					Step[CurrentClient] = CLOSE_PORT;
			}
			else
			if (TCP_Send[CurrentClient].status == TCPIPMGR_TIMEOUT)
			{
			/* VOID, just wait*/
			}
			else	/* any other state, close after a certain time*/
			{
				SendTimeout[CurrentClient]++;
				if(SendTimeout[CurrentClient] > 30) /* 3 sec*/
					Step[CurrentClient] = CLOSE_PORT;
			}
		}

	/***** Port schließen **************************************************/
		if (Step[CurrentClient] == CLOSE_PORT)
		{
			SendTimeout[CurrentClient] = 0;
			TCPclose (&TCP_Close[CurrentClient]);
			/* Status prüfen: */
			if (TCP_Close[CurrentClient].status == TCP_IP_OK)
			{
				/* Port geschlossen, neu öffnen: */
				Step[CurrentClient] = OPEN_PORT;
			}
		} /* if (Step == WAIT_CLOSE_PORT) */

		if (Step[CurrentClient] == WAIT)
		{
			WaitCounter[CurrentClient]++;
			if( WaitCounter[CurrentClient] > 20 )
			{
				Step[CurrentClient] = PREPARE_SEND_DATA;
				WaitCounter[CurrentClient] = 0;
			}
		} /* if (Step == WAIT) */

	} /*for*/
#endif

}
```

### Program Logical/hwconfig (ANSIC, version 0.00.0)

#### hwconfig.c
```c
#ifdef _DEFAULT_INCLUDES
	#include <AsDefault.h>
#endif
/* ===================================================== HEADER FILES ===================================================== */

#include <bur/plc.h>
#include <bur/plctypes.h>
#include <sys_lib.h>
#include <asiomman.h>
#include <brsystem.h>
#include <standard.h>
#include "auxfunc.h"

/* ===================================================== VARAIBLE DECLARATION ==================================================== */

#define ERR_FUB_BUSY 65535
#define MAXHWMODULES (20)
#define ERR_IO_CHECK_NOMODULE (5555)

typedef struct
{
	STRING Name[20];
	UINT HWStatus;
	USINT HWFamily;
	USINT HWUseType;
	USINT HWModuleTyp;
	USINT HWMasterNo;
	USINT HWSlaveNo;
	USINT HWModuleAdr;
	USINT HWSlotNo;
}HW_Info_typ;

_GLOBAL UINT        change_config;                  /* indicates if configuration should be changed */
_GLOBAL UINT        config;                         /* indicates if configuration should be changed */
_GLOBAL USINT       step;                           /* step for the main routine */
_LOCAL  USINT       status_message[128];            /* shows the status of the program */

/* CYCLIC */
_LOCAL  AsIOMMCreate_typ    AsIOMMCreate_Mod;       /* function for creating the new BR module on the target */
_LOCAL  AsIOMMRemove_typ    AsIOMMRemove_Mod;       /* function for removing the BR module on the target */
_LOCAL  AsIOMMCopy_typ      AsIOMMCopy_Mod;         /* function for copying the BR module to a datamodule */
_LOCAL  USINT           error_string[128];

/* shows the last error which occured */
_LOCAL  USINT           error_step;                 /* step where the error occurred */
_LOCAL  UINT            error_status;               /* status of the FBK where the error occured */
_LOCAL  BOOL            error;                      /* shows if an error occurred */
static TON_10ms_typ     WaitTimer;                  /*waits before actually changing config*/
/************************************/

_LOCAL	HWInfo_typ HWInfo_01;

_LOCAL  BOOL            CopyArConfig,CopyIomap,InstallConfig1,InstallConfig2;
_LOCAL  BOOL            next;
_LOCAL	HW_Info_typ		myHWInfo[MAXHWMODULES];
_LOCAL	INT				cnt;
_GLOBAL SINT            IOConfiguration _VAR_RETAIN,NewIOConfig	_VAR_RETAIN;
_GLOBAL SINT 			IOChangeStep	_VAR_RETAIN;

_INIT void InitialisierungsProgramm(void) {
        HWInfo_01.enable = 1;     /* Funktionsblock wird nur ausgeführt
                                   wenn ENABLE <> 0 ist. */
        HWInfo_01.first = 1;      /* Bestimmen des Hardwaremoduls auf dem die
                                   Funktion angewendet werden soll. */
        cnt = 0;
        next = 1;

        InstallConfig1 = 0;
        InstallConfig2 = 0;
        NewIOConfig = 0;
		WaitTimer.IN = 0;
}

_CYCLIC void cyclic( void )
{
	if(next || HWInfo_01.first)
	{
        HWInfo_01.pName = (UDINT) &(myHWInfo[cnt].Name);
        HWInfo(&HWInfo_01);
        myHWInfo[cnt].HWStatus    = HWInfo_01.status;     /* Fehlernummer, 0 ist kein Fehler. */
        myHWInfo[cnt].HWFamily    = HWInfo_01.family;     /* Familienbezeichnung */
        myHWInfo[cnt].HWUseType   = HWInfo_01.usetype;   /* Hardware-Typ */
        myHWInfo[cnt].HWModuleTyp = HWInfo_01.module_typ; /* Typcode des Moduls */
        myHWInfo[cnt].HWMasterNo  = HWInfo_01.master_no;   /* Logische Nummer des IO-Masters, des RIO-Masters bzw.
                                                des CAN-Busses bei CANIO. */
        myHWInfo[cnt].HWSlaveNo   = HWInfo_01.slave_no;     /* Slave Nummer */
        myHWInfo[cnt].HWModuleAdr = HWInfo_01.module_adr;    /* Moduladresse des Hardwaremoduls */
        myHWInfo[cnt].HWSlotNo    = HWInfo_01.slot_no;          /* Steckplatz des Einschub-oder Anpassungsmoduls */

		HWInfo_01.first = 0;
		if(cnt < MAXHWMODULES)
			cnt++;

		if( (HWInfo_01.status == ERR_IO_CHECK_NOMODULE)
		 || (cnt >= MAXHWMODULES)
		  )
		{
			next = 0;
			cnt = 0;
		}
	}

/***********************************************************/

/* change request from pics task (user changes config.)*/

	if(NewIOConfig == 1)
	{
		InstallConfig1 = 1;
		NewIOConfig = 0;
	}
	else
	if(NewIOConfig == 2)
	{
		InstallConfig2 = 1;
		NewIOConfig = 0;
	}

	TON_10ms(&WaitTimer);

	switch (step)
	{
		case 0:
		{
            if(IOChangeStep != 0)
            {
	            if(IOChangeStep == 12)
	            	InstallConfig1 = 1;
	            if(IOChangeStep == 13)
	            	InstallConfig2 = 1;
            	step = 20;
            	IOChangeStep = 0;
            	break;
            }

			if(CopyArConfig)
			{
				CopyArConfig = 0;
				step = 1;
				break;
			}
			if(CopyIomap)
			{
				CopyIomap = 0;
				step = 2;
				break;
			}

			if(InstallConfig1 || InstallConfig2)
			{
				if(WaitTimer.Q)
				{
					WaitTimer.IN = 0;
					step = 5;
					break;
				}
				WaitTimer.IN = 1;
				WaitTimer.PT = 200;
				ShowMessage(128,129,0,INFO,NONE, 1);
				break;
			}
			break;
		}
		case 1:
		{
            AsIOMMCopy_Mod.enable = 1;                            /* enable */
            AsIOMMCopy_Mod.pModuleName = (UDINT) "arconfig";      /* name of the *.br module which has to be removed */
            AsIOMMCopy_Mod.pNewModule = (UDINT) "arcfg2";      /* name of the data module which has to be created */
			AsIOMMCopy_Mod.memType = 2 /*doUSRROM*/;
			AsIOMMCopy_Mod.option = 1;
            /* Call FBK */
            AsIOMMCopy(&AsIOMMCopy_Mod);

            /* Verify status */
            if (AsIOMMCopy_Mod.status == 0 || AsIOMMCopy_Mod.status == iommERR_NOSUCH_MODULE)
            {
                 step = 0;                                          /* next step */
            }
            else
            {
                if (AsIOMMCopy_Mod.status != 0xFFFF)
                {
                    error_step = step;
                    error_status = AsIOMMCopy_Mod.status;
                    step = 100;                                     /* error step */
                    strcpy(error_string, "br_copy_arconfig");
                }
            }
        	break;
		}
		case 2:
		{
            AsIOMMCopy_Mod.enable = 1;                            /* enable */
            AsIOMMCopy_Mod.pModuleName = (UDINT) "iomap";      /* name of the *.br module which has to be removed */
            AsIOMMCopy_Mod.pNewModule = (UDINT) "iomap2";      /* name of the data module which has to be created */
			AsIOMMCopy_Mod.memType = 2 /*doUSRROM*/;
			AsIOMMCopy_Mod.option = 1;
            /* Call FBK */
            AsIOMMCopy(&AsIOMMCopy_Mod);

            /* Verify status */
            if (AsIOMMCopy_Mod.status == 0 || AsIOMMCopy_Mod.status == iommERR_NOSUCH_MODULE)
            {
                 step = 0;                                          /* next step */
            }
            else
            {
                if (AsIOMMCopy_Mod.status != 0xFFFF)
                {
                    error_step = step;
                    error_status = AsIOMMCopy_Mod.status;
                    step = 100;                                     /* error step */
                    strcpy(error_string, "br_copy_iomap");
                }
            }
        	break;
		}

        case 5:     /* CASE 5: Delete "arconfig.br" from target */

            /* Initialize AsIOMMRemove */
            AsIOMMRemove_Mod.enable = 1;                            /* enable */
            AsIOMMRemove_Mod.pModuleName = (UDINT) "arconfig";      /* name of the *.br module which has to be removed */

            /* Call FBK */
            AsIOMMRemove(&AsIOMMRemove_Mod);

            /* Verify status */
            if (AsIOMMRemove_Mod.status == 0)
            {
                step = 6;                                       /* next step */
            }
           else
           {
                if (AsIOMMRemove_Mod.status != 0xFFFF || AsIOMMRemove_Mod.status == iommERR_NOSUCH_MODULE)
                {
                    error_step = step;
                    error_status = AsIOMMRemove_Mod.status;
                    step = 100;                                     /* error step */
                    strcpy(error_string, "br_remove_arconfig");
                }
            }
            break;

        case 6:     /* CASE 6: Delete "iomap.br" from target */

            /* Initialize AsIOMMRemove */
            AsIOMMRemove_Mod.enable = 1;                            /* enable */
            AsIOMMRemove_Mod.pModuleName = (UDINT) "iomap";         /* name of the *.br module which has to be removed */

            /* Call FBK */
            AsIOMMRemove(&AsIOMMRemove_Mod);

            /* Verify status */
            if (AsIOMMRemove_Mod.status == 0 || AsIOMMRemove_Mod.status == iommERR_NOSUCH_MODULE)
            {
                 step = 10;                                       /* next step */
            }
            else
            {
                 if (AsIOMMRemove_Mod.status != 0xFFFF)
                 {
                        error_step = step;
                        error_status = AsIOMMRemove_Mod.status;
                        step = 100;                                 /* error step */
                        strcpy(error_string, "br_remove_iomap");
                 }
            }
            break;

		case 10:
        {
            AsIOMMCreate_Mod.enable = 1;                            /* enable */
			if(InstallConfig1)
			{
	            AsIOMMCreate_Mod.pDataObject = (UDINT) "arcfg1";       /* name of datamodule where the data should be taken from */
    	        AsIOMMCreate_Mod.pNewModule = (UDINT) "arconfig";          /* name of the new *.br module */
    	    }
			else
			{
	            AsIOMMCreate_Mod.pDataObject = (UDINT) "arcfg2";       /* name of datamodule where the data should be taken from */
    	        AsIOMMCreate_Mod.pNewModule = (UDINT) "arconfig";          /* name of the new *.br module */
    	    }
            AsIOMMCreate_Mod.moduleKind = 2 /*config*/;                        /* which type of *.br module should be created */
            AsIOMMCreate_Mod.memType = 2 /*USRROM*/;                           /* where should the *.br module be stored */

            /* Call FBK */
            AsIOMMCreate(&AsIOMMCreate_Mod);

            /* Verify status */
            if (AsIOMMCreate_Mod.status == 0)
            {
                step = 11;                                      /* next step */
            }
            else
            {
                if (AsIOMMCreate_Mod.status != 0xFFFF)
                {
                    error_step = step;
                    error_status = AsIOMMCreate_Mod.status;
                    step = 100;                                     /* error step */
                    strcpy(error_string, "br_create_config");
                }
            }
            break;
         }

		 case 11:
         {
			if(InstallConfig1)
			{
	            IOChangeStep = 12;
         		IOConfiguration = 1;
	        }
	        else
			if(InstallConfig2)
			{
	            IOChangeStep = 13;
         		IOConfiguration = 2;
	        }

            SYSreset(1, 1);                                         /* warm restart for activating new arconfig.br */
            break;
         }

		case 20:
        {

            AsIOMMCreate_Mod.enable = 1;                            /* enable */
			if(InstallConfig1)
			{
	            AsIOMMCreate_Mod.pDataObject = (UDINT) "iomap1";       /* name of datamodule where the data should be taken from */
    	        AsIOMMCreate_Mod.pNewModule = (UDINT) "iomap";          /* name of the new *.br module */
    	    }
			else
			{
	            AsIOMMCreate_Mod.pDataObject = (UDINT) "iomap2";       /* name of datamodule where the data should be taken from */
    	        AsIOMMCreate_Mod.pNewModule = (UDINT) "iomap";          /* name of the new *.br module */
    	    }
            AsIOMMCreate_Mod.moduleKind = 1 /*mapping*/;                        /* which type of *.br module should be created */
            AsIOMMCreate_Mod.memType = 2 /*USRROM*/;                           /* where should the *.br module be stored */

            /* Call FBK */
            AsIOMMCreate(&AsIOMMCreate_Mod);

            /* Verify status */
            if (AsIOMMCreate_Mod.status == 0)
            {
                step = 30;                                      /* next step */
            }
            else
            {
                if (AsIOMMCreate_Mod.status != 0xFFFF)
                {
                    error_step = step;
                    error_status = AsIOMMCreate_Mod.status;
                    step = 100;                                     /* error step */
                    strcpy(error_string, "br_create_iomap");
                }
            }
            break;
         }
		 case 30:
         {
         	if(InstallConfig1)
         		IOConfiguration = 1;
         	else
         	if(InstallConfig2)
         		IOConfiguration = 2;

         	InstallConfig1 = 0;
         	InstallConfig2 = 0;
         	step = 0;
         	IOChangeStep = 0;
            break;
         }

	}/* switch */
}
```

- auxfunc.h (reference to Logical/GlobalIncludes/auxfunc.h)

### Program Logical/udp_nl (ANSIC, version 0.00.0)

- udp.h (reference to Logical/GlobalIncludes/udp.h)

#### udp.c
```c
#ifdef _DEFAULT_INCLUDES
	#include <AsDefault.h>
#endif
/*
                             *******************
******************************* C SOURCE FILE *******************************
**                           *******************                           **
**                                                                         **
** project  : Jet3                                                         **
** filename : UDP.C                                                        **
** version  : 1.00                                                         **
** date     : 24.09.2010                                                   **
**                                                                         **
*****************************************************************************
** Abstract                                                                **
** ========                                                                **
** implements an udp client/server                                         **
**                                                                         **
** Copyright (c) 2010, Krause-Biagosch GmbH                                **
** All rights reserved.                                                    **
**                                                                         **
*****************************************************************************
VERSION HISTORY:
----------------
Version     : 1.00
Date        : 24.09.2010
Revised by  : Herbert Aden
Description : Original version. Based on XJet Version

*/

#define _UDP_C

/****************************************************************************/
/**                                                                        **/
/**                           INCLUDE FILES                                **/
/**                                                                        **/
/****************************************************************************/
#include "udp.h"
#include "auxfunc.h"

/****************************************************************************/
/**                                                                        **/
/**                       DEFINITIONS AND MACROS                           **/
/**                                                                        **/
/****************************************************************************/

/****************************************************************************/
/**                                                                        **/
/**                          LOCAL FUNCTIONS                               **/
/**                                                                        **/
/****************************************************************************/

/*
 * copies the last n chars from src to dest, if n>strlen(src) the complete
 * src string will be copied
 * returns the actual no of chars copied
 */
int strendcpy(char *dest,const char *src,int n)
{
	const char *p1;
	int srclen = strlen(src);
	int offs = srclen - n;
	int res = srclen;

	if(offs > 0)
	{
		p1 = &src[offs];
		strcpy(dest,p1);
		res = n;
	}
	else
		strcpy(dest,src);

	return res;
}

/****************************************************************************/
/* Parser */
/****************************************************************************/
void Parse(char *buf)
{
	char *pctmp;
	char token[MAXTOKENS][MAXTOKENLENGTH];
	int i = 0;
/* erstmal alle Tokens initialisieren*/
	for(i=0;i<MAXTOKENS;i++)
		strcpy(token[i],"-");

	strncpy(DebugRecStr,buf,DEBUGSTRSIZE-1);
	DebugRecStr[DEBUGSTRSIZE-1] = '\0';

	i = 0;
	pctmp = strtok(&buf[0],(char *)";");
	do
	{
		if(pctmp != NULL)
		{
			strncpy(token[i],pctmp,MAXTOKENLENGTH-1);
			token[i][MAXTOKENLENGTH-1] = '\0';
			i++;
		}
		pctmp = strtok(NULL,(char *)";");
	}
	while (pctmp != NULL && i<MAXTOKENS);

	if( STREQN(&buf[0],"la paloma",9)
	 || STREQN(&buf[0],"La Paloma",9)
	 || STREQN(&buf[0],"La paloma",9)
	 || STREQN(&buf[0],"la Paloma",9)
	  )
		SendTestAnswer = TRUE;
	else
	if( i > 2 )
	{
/* Netlink Kommandos */
		if(STREQN(token[0],"PERFOXXL",8))
		{
			if(i > 3)
			{
				if(STREQN(token[1],"NEXTJOB",7))
				{
/*
token2 -> job id
token3 -> plate type
token4 -> next plate type
token5 -> plateconfig
 */
					int tmpPlateType = atoi((UDINT)token[3]);
					strcpy(tmpID,token[2]);
					if(!START)
						SendJobAnswer = SEND_MACHINE_NOT_STARTED;
					else
					if(PlateAtAdjustedPosition.present && (STREQN(PlateAtAdjustedPosition.ID,"???",3)))
					{
						strcpy(PlateAtAdjustedPosition.ID,tmpID);
						SendJobAnswer = SEND_OK;
					}
					else
					if(PlateAtFeeder.present && (STREQN(PlateAtFeeder.ID,"???",3)))
					{
						strcpy(PlateAtFeeder.ID,tmpID);
						SendJobAnswer = SEND_OK;
						if( (tmpPlateType == atoi((UDINT)token[4]))
						 && !PlateToDo.present
						  )
						{
							PlateToDo.present = TRUE;
							PlateToDo.PlateType = tmpPlateType;
							PlateToDo.NextPlateType = 0;
							PlateToDo.PlateConfig = PlateAtFeeder.PlateConfig;
							strcpy(PlateToDo.ID,"???");
						}
					}
					else
					if(PlateToDo.present)
					{
						if(STREQN(PlateToDo.ID,"???",3))
						{
							strcpy(PlateToDo.ID,tmpID);
							if(!ManualMode)
								PlateToDo.NextPlateType = atoi((UDINT)token[4]);
							SendJobAnswer = SEND_OK;
						}
						else
							SendJobAnswer = SEND_BUFFER_FULL;
					}
					else
					if((tmpPlateType > 0) && (tmpPlateType < MAXPLATETYPES))
					{
						USINT PlateTypeToCheck;
						if((GlobalParameter.TrolleyLeft == 0) || (GlobalParameter.TrolleyLeft >= MAXTROLLEYS))
							GlobalParameter.TrolleyLeft = 1;

						if(ManualMode)
							PlateTypeToCheck = PlateType; /* manual mode platetype selected by user */
						else
							PlateTypeToCheck = Trolleys[GlobalParameter.TrolleyLeft].PlateType;

						if(tmpPlateType != PlateTypeToCheck)
							SendJobAnswer = SEND_PLATE_NOT_LOADED;
						else
						{
							PlateToDo.present = TRUE;
							PlateToDo.PlateType = tmpPlateType;
							strcpy(PlateToDo.ID,tmpID);
							if(STREQ(token[5],"10"))
								PlateToDo.PlateConfig = LEFT;
							if(STREQ(token[5],"02"))
								PlateToDo.PlateConfig = RIGHT;
							if(STREQ(token[5],"12"))
								PlateToDo.PlateConfig = BOTH;
							if(STREQ(token[5],"3") || STREQ(token[5],"30"))
								PlateToDo.PlateConfig = PANORAMA;
							if(STREQ(token[5],"4") || STREQ(token[5],"40"))
								PlateToDo.PlateConfig = BROADSHEET;

							if(!ManualMode)
								PlateToDo.NextPlateType = atoi((UDINT)token[4]);

							SendJobAnswer = SEND_OK;
						}
					}
					else
						SendJobAnswer = SEND_PLATE_NOT_LOADED;
				}
			}
		}
		else
/* LSJet Kommandos */
		if(STREQN(token[0],"JET",3))
		{
			if(i == 3)
			{
				if(STREQN(token[2],"\r\n",2))
				{
					if( STREQN(token[1],"START",5))
					{
						START = TRUE;
						SendJetStartOK = TRUE;
					}
					else
					if( STREQN(token[1],"STOP",4))
					{
						START = FALSE;
						SendJetStopOK = TRUE;
					}
					else
					if( STREQN(token[1],"REFERENCE",9))
					{
						ReferenceStart = TRUE;
						SendJetRefOK = TRUE;
					}
					else
					if( STREQN(token[1],"CONTROLVOLTAGE",14))
					{
						SendJetControlvoltageOK = TRUE;
					}
					else
					if( STREQN(token[1],"ANSWEROK",8))
					{
						gAbfrageOK = TRUE;
						AlarmBitField[15] = FALSE; /* Trolley leer */
						AlarmBitField[26] = FALSE; /* Ausrichtfehler */
						AlarmBitField[28] = FALSE; /* Vakuumfehler Aufnahme */
						AlarmBitField[29] = FALSE; /* Vakuumfehler Übergabe */
					}
					else
					if( STREQN(token[1],"ANSWERCANCEL",12))
					{
						gAbfrageCancel = TRUE;
					}
					else
					if( STREQN(token[1],"CLEARMACHINE",12))
					{
						gClearLinePressed = TRUE;
					}
					else
					if( STREQN(token[1],"STEPWEDGE",9))
					{
/*
						Expose_Param.StepwedgeExposure = TRUE;
						SendStepwedgeOK = TRUE;
*/
					}
				}
			}
		}
		else
		if( STREQN(token[0],"CLEARMACHINE",12))
		{
			gClearLinePressed = TRUE;
		}
	}
}

/****************************************************************************/
/* INIT Teil*/
/****************************************************************************/
_INIT void init_UDP(void)
{
	strcpy(&buffer[0], "nothing sent");             /* Initialize the buffer */
	strcpy(&receivebuffer[0], "nothing received");             /* Initialize the buffer */
	counter = 0;
	UDPStep = 0;
	UDPRcvStep = 0;
	CounterMax = 5;
	StatusRequestTimeout.IN = FALSE;
	StatusRequestTimeout.PT = 1200;
	StatusRequestTimer.IN = FALSE;
	SendStatusInterval = 30;
	StatusRequestTimer.PT = SendStatusInterval;
	PlateAtFeeder.present = FALSE;
	PlateAtFeeder.PlateType = 0;
	strcpy(PlateAtFeeder.ID,"");
	PlateAtFeeder.ErrorCode = 0;
	PlateAtFeeder.Status = 0;

	PlateToDo = PlateAtFeeder;
	PlateToDo.PlateConfig = BOTH;
	PlateAtAdjustedPosition = PlateAtFeeder;
}

/****************************************************************************/
/* CYCLIC Teil*/
/****************************************************************************/
_CYCLIC void cyclic_UDP(void)
{
	TON_10ms(&StatusRequestTimeout);

	if( StatusRequestTimeout.Q )
	{
		StatusRequestTimeout.IN = FALSE;
	}

/* Statusrequest alle 1 sec triggern*/
	MachineOnlineEdgeR.CLK = START;
	R_TRIG(&MachineOnlineEdgeR);
	MachineOfflineEdgeR.CLK = !START;
	R_TRIG(&MachineOfflineEdgeR);
	if(MachineOnlineEdgeR.Q || MachineOfflineEdgeR.Q)
		SendStatusRequest = TRUE;

	StatusRequestTimer.IN = !SendStatusRequest;
	StatusRequestTimer.PT = SendStatusInterval;
	TON_10ms(&StatusRequestTimer);

	switch (UDPStep)
	{
		case 0:
		{

			if(
			    SendStatusRequest
			 || SendJobStates
			 || (SendJobAnswer != 0)
			 )
			{
				UDPStep = 10;
			}
			else
			if(StatusRequestTimer.Q)
			{
				StatusRequestTimer.IN = FALSE;
				{
					SendStatusRequest = TRUE;
					SendJobStates = TRUE;
				}
			}

			break;
		}

		case 10:
		{
			UDPopen_1.enable = TRUE;
			UDPopen_1.port = 60000;
			UDPopen_1.pIfAddr = NULL;
			UdpOpen(&UDPopen_1);
			if(UDPopen_1.status == 0)
				UDPStep = 20;
			if(UDPopen_1.status == udpERR_ALREADY_EXIST)
			{
				UDPclose_1.enable = TRUE;             /* Enables the FBK */
				UDPclose_1.ident = UDPopen_1.ident;
				UdpClose(&UDPclose_1);        /* Close the connection */
			}
			break;
		}
		case 20:
		{
			int length = 0;

			if(SendJobAnswer != 0)
			{
				switch (SendJobAnswer)
				{
					case SEND_OK:
					{
						strcpy(buffer,"PERFOXXL;NEXTJOB;");
						strcat(buffer,tmpID);
						strcat(buffer,";ACCEPTED");
						break;
					}
					case SEND_BUFFER_FULL:
					{
						strcpy(buffer,"PERFOXXL;NEXTJOB;");
						strcat(buffer,tmpID);
						strcat(buffer,";BUSY");
						break;
					}
					case SEND_MACHINE_NOT_STARTED:
					{
						strcpy(buffer,"PERFOXXL;NEXTJOB;");
						strcat(buffer,tmpID);
						strcat(buffer,";NOTSTARTED");
						break;
					}
					case SEND_PLATE_NOT_LOADED:
					{
						strcpy(buffer,"PERFOXXL;NEXTJOB;");
						strcat(buffer,tmpID);
						strcat(buffer,";WRONGPLATETYPE");
						break;
					}
					default:
					{
						strcpy(buffer,"PERFOXXL;NEXTJOB;");
						strcat(buffer,tmpID);
						strcat(buffer,";ERROR");
						break;
					}
				}
				strcat(buffer,"\r\n");
				length = strlen(buffer);
				SendJobAnswer = 0;
			}
			else
			if(SendStatusRequest)
			{
				SendStatusRequest = FALSE;
/*
				strcpy(buffer,"alive");
				strcat(buffer,"\r\n");
				length = strlen(buffer);
*/
			}
			else
			if(SendTestAnswer)
			{
				SendTestAnswer = FALSE;
				strcpy(buffer,"einmal muss es vohorbei sein...");
				strcat(buffer,"\r\n");
				length = strlen(buffer);
			}
			else
			if(SendJobStates)
			{
				SendJobStates = FALSE;
			}
/*
			else
			if(SendJobStates)
			{
				int i=0;
				strcpy(buffer,"PLATESTATE;");
				for(i=0;i<=1;i++)
				{
					if(PlateToDo[i].present)
					{
						strcat(buffer,PlateToDo[i].ID);
						strcat(buffer,STR_PLATESTATE_RESERVED);
					}
				}
				for(i=0;i<=1;i++)
				{
					if(PlateAtFeeder[i].present)
					{
						strcat(buffer,PlateAtFeeder[i].ID);
						strcat(buffer,STR_PLATESTATE_FEEDER);
					}
				}
				for(i=0;i<=1;i++)
				{
					if(PlateAtShuttle[i].present)
					{
						strcat(buffer,PlateAtShuttle[i].ID);
						strcat(buffer,STR_PLATESTATE_SHUTTLE);
					}
				}
				if(PlateAtDropPosition.present)
				{
					strcat(buffer,PlateAtDropPosition.ID);
					strcat(buffer,STR_PLATESTATE_TABLE);
				}
				if(PlateAtAdjustedPosition.present)
				{
					strcat(buffer,PlateAtAdjustedPosition.ID);
					switch (PlateAtAdjustedPosition.Status)
					{
						case PLATESTATE_ALIGNED:
						{
							strcat(buffer,STR_PLATESTATE_ALIGNED);
							break;
						}
						case PLATESTATE_IMAGING:
						{
							strcat(buffer,STR_PLATESTATE_IMAGING);
							break;
						}
						case PLATESTATE_DELOADING:
						{
							strcat(buffer,STR_PLATESTATE_DELOADING);
							break;
						}
						default:
						{
							strcat(buffer,STR_PLATESTATE_ALIGNED);
							break;
						}
					}
				}
				if(PlateOnConveyorBelt.present)
				{
					strcat(buffer,PlateOnConveyorBelt.ID);
					strcat(buffer,STR_PLATESTATE_CONVEYORBELT);
				}

				for(i=0;i<FAILEDPLATESARRAYSIZE;i++)
				{
					if(FailedPlate[i].present)
					{
						strcat(buffer,FailedPlate[i].ID);
						switch (FailedPlate[i].Status)
						{
							case PLATESTATE_FEEDERVAC_FAIL:
							{
								strcat(buffer,STR_PLATESTATE_FEEDERVAC_FAIL);
								break;
							}
							case PLATESTATE_SHUTTLEVAC_FAIL:
							{
								strcat(buffer,STR_PLATESTATE_SHUTTLEVAC_FAIL);
								break;
							}
							case PLATESTATE_ALIGN_FAIL:
							{
								strcat(buffer,STR_PLATESTATE_ALIGN_FAIL);
								break;
							}
							default:
							{
								strcat(buffer,STR_GENERAL_ERROR);
								break;
							}
						}

						ClearStation(&FailedPlate[i]);
					}
				}

				if(strlen(buffer) <= strlen("PLATESTATE;"))
					strcat(buffer,"NO PLATES;");

				strcat(buffer,"\r\n");
				length = strlen(buffer);
				SendJobStates = FALSE;
			}
*/
/* Add more send commands here*/

			if( (length > 0) && (length < SENDBUFSIZE) )
			{
				UDPsend_1.enable = TRUE;             /* Enables the FBK */
				UDPsend_1.ident = UDPopen_1.ident; /* Copy the Ident number */
				UDPsend_1.pData = (UDINT)&buffer[0];/* Address of the buffer */
				UDPsend_1.datalen = length;
				UDPsend_1.pHost = (UDINT) &RemoteIP[0];
				UDPsend_1.port = 60000;     /* Port number of the receiver */
				UDPStep = 35;
				strncpy(DebugSendStr,buffer,DEBUGSTRSIZE-1);
				DebugSendStr[DEBUGSTRSIZE-1] = '\0';
			}
			else
			{
				UDPStep = 40;
			}
			break;
		}

		case 35:
		{
			UdpSend(&UDPsend_1);        /* Sends the data to the member */
			if(UDPsend_1.status == 0)
			{
				UDPStep = 40;
				strcpy(buffer,"");
			}
			break;
		}

		case 40:
		{
			UDPclose_1.enable = 1;             /* Enables the FBK */
			UDPclose_1.ident = UDPopen_1.ident;
			UdpClose(&UDPclose_1);        /* Close the connection */
			if(UDPclose_1.status == 0)
				UDPStep = 0;
			counter = 0;
			break;
		}
	}

	switch (UDPRcvStep)
	{

		case 0:
		{
			UDPopen_Rcv.enable = TRUE;
			UDPopen_Rcv.port = 60001;
			UDPopen_Rcv.pIfAddr = NULL;
			UdpOpen(&UDPopen_Rcv);
			if(UDPopen_Rcv.status == 0)
				UDPRcvStep = 20;
			if(UDPopen_Rcv.status == udpERR_ALREADY_EXIST)
			{
				UDPclose_1.enable = TRUE;             /* Enables the FBK */
				UDPclose_1.ident = UDPopen_Rcv.ident;
				UdpClose(&UDPclose_1);        /* Close the connection */
			}

			break;
		}
		case 20:
		{
			STRING oldRemoteIP[20];
			strcpy(oldRemoteIP,RemoteIP);

			UDPreceive_1.enable = TRUE;             /* Enables the FBK */
			UDPreceive_1.ident = UDPopen_Rcv.ident; /* Copy the Ident number */
			UDPreceive_1.pData = (UDINT)&receivebuffer[0];/* Address of the buffer */
			UDPreceive_1.datamax = sizeof(receivebuffer)-1;   /* Size of the buffer */
			UDPreceive_1.pIpAddr = (UDINT) &RemoteIP[0];

			UdpRecv(&UDPreceive_1);        /* receives data from the member */

			remotePort = UDPreceive_1.port;

			if( UDPreceive_1.status == 0 )
			{
				if( !STREQ(oldRemoteIP,RemoteIP)
				 && (RemoteIP[0] == '1')
				 && (RemoteIP[1] == '9')
				 && (RemoteIP[2] == '2')
				 && (RemoteIP[3] == '.')
				 )
					saveRemoteIP = TRUE;
				receivebuffer[UDPreceive_1.recvlen] = 0;
				Parse(receivebuffer);

			} /* if status==0 */
			break;
		}
	}

}

/****************************************************************************/
/**                                                                        **/
/**                                 EOF                                    **/
/**                                                                        **/
/****************************************************************************/
```

- glob_var.h (reference to Logical/GlobalIncludes/glob_var.h)

- auxfunc.h (reference to Logical/GlobalIncludes/auxfunc.h)

### Package Logical/Datenobj - Datenobjekte

### Data object Logical/Datenobj/ioimgcfg (Simple, version 0.00.0)

#### ioimgcfg.dat
```
; von Automation Studio generierte Datei.
; Jede Änderung des Dateinhaltes deaktiviert
; die weitere automatische Aktualisierung dieser Datei durch Automation Studio!
```

### Data object Logical/Datenobj/can_tab (Simple, version 0.00.0)

#### can_tab.dat
```
;~~~~~~~~~~~~~~~~~~~~~~~~~~~~~~~~~~~~~~~~~~~~~~~~~~~~~~~~~~~~~~~~~~~~~~~~~~~
;  Datenmodul für CAN IDs
;
;~~~~~~~~~~~~~~~~~~~~~~~~~~~~~~~~~~~~~~~~~~~~~~~~~~~~~~~~~~~~~~~~~~~~~~~~~~~

;       +------------------------------------- can_id [long]
;       |                                +---- pv_name [32 byte]
;       |                                |     Info [long] (bit0=0:read|bit0=1:write)-+
;       |                                |     event_pv[32 byte]-----------+          |
;       |                                |                                 |          |
;|-long-|  |---------- 31 char ----------|   |---------- 31 char ----------|   |-long-|
;
;Nordac FU IDs
;
$00000607,"Can_FU.InitRes                 ","Can_FU.InitResEv               ",$00000000
$000000dd,"Can_FU.InitReq                 ","Can_FU.InitReqEv               ",$00000001
$00000371,"Can_FU.StatRes                 ","Can_FU.StatResEv               ",$00000000
$00000295,"Can_FU.SteuReq                 ","Can_FU.SteuReqEv               ",$00000001
$0000044d,"Can_FU.ParaReq                 ","Can_FU.ParaReqEv               ",$00000001
$00000529,"Can_FU.ParaRes                 ","Can_FU.ParaResEv               ",$00000000
;
;
;
;
;~~~ Ende ~~~~~~~~~~~~~~~~~~~~~~~~~~~~~~~~~~~~~~~~~~~~~~~~~~~~~~~~~~~~~~~~~~~~~~~~~~~~~~
```

### Data object Logical/Datenobj/do_ima (Simple, version 0.00.0)

#### do_ima.dat
```
;------------------------------------------------------------------------------------------------
;AsIMA Konfigurations-Datenobjekt für STATION1
;------------------------------------------------------------------------------------------------

"[ROUTING_PATH]"    ;Sektionsname muss mit Klammern umrahmt werden und ist frei wählbar
"/SECTION=INTERFACE";definiert Sektionsart
"/CN=SL1.SS1.IF1.3" ;Routingpfad zum Server (CANModul Slot1 Schnittstelle 1 Interface 1 zu
                    ;Knotennummer 3) ACHTUNG:
                    ;Knotennummer muss in HEXADEZIMAL angegeben werden !
;===============================================================================================
"[PV_LIST_1]"       ;Sektionsname muss mit Klammern umrahmt werden und ist frei wählbar
"/SECTION=PV"       ;definiert Sektionsart
"/CONPV=bluefin:EnablePVComm /CONVAL=1 /MINT=0 /MAXT=0"     ;optional, gültig für ganze Sektion
"/SV=READ /CLNTPV=bluefin:OldXMLBuffer /SERVPV=xml:XMLBuffer /EVPV=bluefin:byte_link_cnt"  ;PV-Dienst
"/SV=WRITE /CLNTPV=bluefin:DataLock /SERVPV=xml:DataLock"
;===============================================================================================
"[PV_LIST_2]"       ;Sektionsname muss mit Klammern umrahmt werden und ist frei wählbar
"/SECTION=PV"       ;definiert Sektionsart
"/SV=READ /CLNTPV=bluefin:CAN_EGM1 /SERVPV=NoError"  ;PV-Dienst
"/SV=READ /CLNTPV=bluefin:CAN_EGM2 /SERVPV=Ready"  ;PV-Dienst
"/SV=READ /CLNTPV=bluefin:BFVERSION  /SERVPV=gVERSION"  ;PV-Dienst
;===============================================================================================
```

### Data object Logical/Datenobj/do_vcp (Simple, version 0.00.0)

#### do_vcp.dat
```
;------------------------------------------------------------------------------------------------
;AsIMA Konfigurations-Datenobjekt für STATION1
;------------------------------------------------------------------------------------------------

"[ROUTING_PATH]"    ;Sektionsname muss mit Klammern umrahmt werden und ist frei wählbar
"/SECTION=INTERFACE";definiert Sektionsart
"/CN=SL1.SS1.IF1.3" ;Routingpfad zum Server (CANModul Slot1 Schnittstelle 1 Interface 1 zu
                    ;Knotennummer 3) ACHTUNG:
                    ;Knotennummer muss in HEXADEZIMAL angegeben werden !
;===============================================================================================
"[PV_LIST_1]"       ;Sektionsname muss mit Klammern umrahmt werden und ist frei wählbar
"/SECTION=PV"       ;definiert Sektionsart
"/CONPV=bluefin:EnablePVComm /CONVAL=1 /MINT=0 /MAXT=0"     ;optional, gültig für ganze Sektion
"/SV=READ /CLNTPV=bluefin:XMLBuffer /SERVPV=xml:XMLBuffer /EVPV=bluefin:byte_link_cnt"  ;PV-Dienst
"/SV=WRITE /CLNTPV=bluefin:DataLock /SERVPV=xml:DataLock"
;===============================================================================================
"[PV_LIST_2]"       ;Sektionsname muss mit Klammern umrahmt werden und ist frei wählbar
"/SECTION=PV"       ;definiert Sektionsart
"/SV=READ /CLNTPV=bluefin:CAN_EGM1 /SERVPV=NoError"  ;PV-Dienst
"/SV=READ /CLNTPV=bluefin:CAN_EGM2 /SERVPV=Ready"  ;PV-Dienst
"/SV=READ /CLNTPV=bluefin:CAN_VCP  /SERVPV=VCP_OK"  ;PV-Dienst
"/SV=READ /CLNTPV=bluefin:BFVERSION  /SERVPV=gVERSION"  ;PV-Dienst
;===============================================================================================
```

### Data object Logical/Datenobj/do_xsold (Simple)

#### do_xsold.dat
```
;------------------------------------------------------------------------------------------------
;AsIMA Konfigurations-Datenobjekt für STATION1
;------------------------------------------------------------------------------------------------

"[ROUTING_PATH]"    ;Sektionsname muss mit Klammern umrahmt werden und ist frei wählbar
"/SECTION=INTERFACE";definiert Sektionsart
"/CN=SL1.SS1.IF1.3" ;Routingpfad zum Server (CANModul Slot1 Schnittstelle 1 Interface 1 zu
                    ;Knotennummer 3) ACHTUNG:
                    ;Knotennummer muss in HEXADEZIMAL angegeben werden !
;===============================================================================================
"[PV_LIST_1]"       ;Sektionsname muss mit Klammern umrahmt werden und ist frei wählbar
"/SECTION=PV"       ;definiert Sektionsart
"/CONPV=bluefin:EnablePVComm /CONVAL=1 /MINT=0 /MAXT=0"     ;optional, gültig für ganze Sektion
"/SV=READ /CLNTPV=bluefin:OldXMLBuffer /SERVPV=xml:XMLBuffer /EVPV=bluefin:byte_link_cnt"  ;PV-Dienst
"/SV=WRITE /CLNTPV=bluefin:DataLock /SERVPV=xml:DataLock"
;===============================================================================================
"[PV_LIST_2]"       ;Sektionsname muss mit Klammern umrahmt werden und ist frei wählbar
"/SECTION=PV"       ;definiert Sektionsart
"/SV=READ /CLNTPV=bluefin:CAN_EGM1 /SERVPV=NoError"  ;PV-Dienst
"/SV=READ /CLNTPV=bluefin:CAN_EGM2 /SERVPV=Ready"  ;PV-Dienst
"/SV=READ /CLNTPV=bluefin:CAN_VCP  /SERVPV=VCP_OK"  ;PV-Dienst
"/SV=READ /CLNTPV=bluefin:BFVERSION  /SERVPV=gVERSION"  ;PV-Dienst
;===============================================================================================
```

- Visualisation Logical/Visualisierung (not shown)

### Package Logical/Exposer - Belichter tasks

### Package Logical/Exposer/Hardware - Ansteuerung EA, Motoren etc

### Program Logical/Exposer/Hardware/motoren (ANSIC, version 1.00.0) - Referenzfahrt der Motoren

#### motorref.c
```c
#ifdef _DEFAULT_INCLUDES
	#include <AsDefault.h>
#endif
/*
                             *******************
******************************* C SOURCE FILE *******************************
**                           *******************                           **
**                                                                         **
** project  : LS JET II                                                    **
** filename : MOTORREF.C                                                   **
** version  : 1.11                                                         **
** date     : 24.01.2008                                                   **
**                                                                         **
*****************************************************************************
** Abstract                                                                **
** ========                                                                **
** Sequence for reference cycle of motors                                  **
**                                                                         **
**                                                                         **
** Copyright (c) 2006, Krause-Biagosch GmbH                                **
** All rights reserved.                                                    **
**                                                                         **
*****************************************************************************
VERSION HISTORY:
----------------
Version     : 1.00
Date        : 05.09.2002
Revised by  : Herbert Aden
Description : Original version.

Version     : 1.10
Date        : 07.11.2006
Revised by  : Herbert Aden
Description : -Code review, style improvement

Version     : 1.11
Date        : 24.01.2008
Revised by  : Herbert Aden
Description : Added ANSW0 command at reference to make sure, the motor will
              not send unexpectedly

*/
#define _MOTORREF_C_SRC

/****************************************************************************/
/**                                                                        **/
/**                           INCLUDE FILES                                **/
/**                                                                        **/
/****************************************************************************/
#include <string.h>
#include "asstring.h"
#include "glob_var.h"
#include "in_out.h"
#include "auxfunc.h"
#include "motorfunc.h"

/****************************************************************************/
/**                                                                        **/
/**                       DEFINITIONS AND MACROS                           **/
/**                                                                        **/
/****************************************************************************/

#define TIMEOUT		10	/*timeout for moving to obstacle*/
#define WAITTIME	5	/*Waittime after M cmd for moving off ref position */

/****************************************************************************/
/**                                                                        **/
/**                      TYPEDEFS AND STRUCTURES                           **/
/**                                                                        **/
/****************************************************************************/
/* NONE */

/****************************************************************************/
/**                                                                        **/
/**                      PROTOTYPES OF EXTERNAL FUNCTIONS                  **/
/**                                                                        **/
/****************************************************************************/
extern void MotorPicture(void);
extern void MotorManual(void);
extern void MotorTarget(void);
extern void MotorStop(void);

/****************************************************************************/
/**                                                                        **/
/**                      PROTOTYPES OF LOCAL FUNCTIONS                     **/
/**                                                                        **/
/****************************************************************************/
/* NONE */

/****************************************************************************/
/**                                                                        **/
/**                      EXPORTED VARIABLES                                **/
/**                                                                        **/
/****************************************************************************/
/* NONE */

/****************************************************************************/
/**                                                                        **/
/**                           GLOBAL VARIABLES                             **/
/**                                                                        **/
/****************************************************************************/
_GLOBAL   UINT                ConveyorBeltOn;

/****************************************************************************/
/**                                                                        **/
/**                      TASK-LOCAL VARIABLES                              **/
/**                                                                        **/
/****************************************************************************/
_LOCAL    INT                 CurrentMotor;

/****************************************************************************/
/**                                                                        **/
/**                    MODULE-LOCAL VARIABLES                              **/
/**                                                                        **/
/****************************************************************************/
static    USINT               OldPriority[MAXMOTORS];
static    UDINT               OldPositionWindow[MAXMOTORS];
static    UDINT               Timeouts[MAXMOTORS];

/****************************************************************************/
/**                                                                        **/
/**                          EXPORTED FUNCTIONS                            **/
/**                                                                        **/
/****************************************************************************/
/* NONE */

/****************************************************************************/
/**                                                                        **/
/**                          LOCAL FUNCTIONS                               **/
/**                                                                        **/
/****************************************************************************/

/****************************************************************************/
/** Init function, executed once at startup                                **/
/****************************************************************************/
_INIT void init(void)
{
	int i;
	for(i=0;i<MAXMOTORS;i++)
		Timeouts[i] = 0;
	loadMotorData = TRUE;
	CurrentMotor = 1;
}

_CYCLIC void c(void)
{

	if(loadMotorData || loadParameterData) return;

	if( GlobalParameter.DeloaderTurnStation == NO_DELOADER )
	{
		Motors[DELOADER_HORIZONTAL].Error = FALSE;
		Motors[DELOADER_HORIZONTAL].Moving = FALSE;
		Motors[DELOADER_HORIZONTAL].ReferenceOk = TRUE;
	}

	if( GlobalParameter.DeloaderTurnStation != DELOADER_AND_TURNSTATION )
	{
		Motors[DELOADER_TURN].Error = FALSE;
		Motors[DELOADER_TURN].Moving = FALSE;
		Motors[DELOADER_TURN].ReferenceOk = TRUE;
	}

	if( GlobalParameter.FlexibleFeeder == FALSE)
	{
		Motors[FEEDER_HORIZONTAL].Error = FALSE;
		Motors[FEEDER_HORIZONTAL].Moving = FALSE;
		Motors[FEEDER_HORIZONTAL].ReferenceOk = TRUE;
	}

/* call external functions */
	MotorManual();   /* in motorman.c */
	MotorTarget();   /* in motortarget.c */
	MotorStop();     /* in motorstop.c */

/*Reference in a loop for all motors*/
	switch (Motors[CurrentMotor].ReferenceStep)
	{
		case 0:
		{
			if(   (Motors[CurrentMotor].StartRef == TRUE)
			   && (Motors[CurrentMotor].Error    == FALSE) )
			   Motors[CurrentMotor].ReferenceStep = 102;
			break;
		}
/*V5.04 send ANSW0 to avoid asynchronous answers from motor */
		case 102:
		{
			if( SendMotorCmd(CurrentMotor, CMD_NOANSW, FALSE, 0L) )
			{
				Motors[CurrentMotor].ReferenceStep = 103;
			}
			break;
		}
		case 103:
		{
			if( SendMotorCmd(CurrentMotor, CMD_COMPATIBLE, FALSE, 0L) )
			{
				Motors[CurrentMotor].ReferenceStep = 1;
			}
			break;
		}

		case 1:
		{
/* enable Motor */
			if( SendMotorCmd(CurrentMotor, CMD_ENABLE, FALSE, 0L) )
			{
				OldPriority[CurrentMotor] = Motors[CurrentMotor].Parameter.Priority;
				OldPositionWindow[CurrentMotor] = Motors[CurrentMotor].Parameter.PositionWindow;
				Motors[CurrentMotor].Parameter.Priority = 1;
				Motors[CurrentMotor].Parameter.PositionWindow = 50;
				Motors[CurrentMotor].ReferenceStep = 2;
			}
			break;
		}
		case 2:
		{
/*SOR0*/
			if( SendMotorCmd(CurrentMotor, CMD_SERIAL, FALSE, 0L) )
			{
				Motors[CurrentMotor].ReferenceStep = 3;
			}
			break;
		}

		case 3:
		{
/*stop motor*/
			if( SendMotorCmd(CurrentMotor, CMD_STOP, FALSE, 0L) )
			{
				if(CurrentMotor == CONVEYORBELT)
					ConveyorBeltOn = FALSE;

				if(CurrentMotor == ADJUSTER || CurrentMotor == CONVEYORBELT)
					Motors[CurrentMotor].ReferenceStep = 20;
				else
					Motors[CurrentMotor].ReferenceStep = 4;
			}
			break;
		}

		case 4:
		{
			if( SendMotorCmd(CurrentMotor, CMD_ACCELERATION, TRUE, Motors[CurrentMotor].Parameter.ReferenceAcceleration) )
			{
				Motors[CurrentMotor].ReferenceStep = 5;
			}
			break;
		}
		case 5:
		{
			if( SendMotorCmd(CurrentMotor, CMD_CONT_CURRENT, TRUE, Motors[CurrentMotor].Parameter.ReferenceContCurrent) )
			{
				Motors[CurrentMotor].ReferenceStep = 10;
			}
			break;
		}
		case 10:
		{
			if( SendMotorCmd(CurrentMotor, CMD_PEAK_CURRENT, TRUE, Motors[CurrentMotor].Parameter.ReferencePeekCurrent) )
			{
				Motors[CurrentMotor].ReferenceStep = 11;
			}
			break;
		}
		case 11:
		{
			if( SendMotorCmd(CurrentMotor, CMD_PROPFACT, TRUE, Motors[CurrentMotor].Parameter.ReferencePropFact) )
			{
				Motors[CurrentMotor].ReferenceStep = 12;
			}
			break;
		}
		case 12:
		{
			if( SendMotorCmd(CurrentMotor, CMD_INTFACT, TRUE, Motors[CurrentMotor].Parameter.ControllerIFact) )
			{
/* HA 20160120 V1.40 added Paletteloading
 * Paperremove vertical: if sensor "up" gives signal, go to step 20
 */
				if( GlobalParameter.EnablePaletteLoading && (CurrentMotor == PAPERREMOVE_VERTICAL))
				{
					if(In_PaperRemoveUp)
					{
						Motors[CurrentMotor].ReferenceStep = 20;
						Timeouts[CurrentMotor] = 0;
						Motors[CurrentMotor].timeout=0;
						break;
					}
				}
				Motors[CurrentMotor].ReferenceStep=13;
				Motors[CurrentMotor].timeout=0;
				Timeouts[CurrentMotor] = 0;
			}
			break;
		}

		case 13:
		{
			DINT	tmpval;
			tmpval = (-1L) * labs(Motors[CurrentMotor].Parameter.ReferenceSpeed);
			if( SendMotorCmd(CurrentMotor, CMD_MOVE_AT, TRUE, tmpval) )
			{
				Motors[CurrentMotor].ReferenceStep = 15;
				Motors[CurrentMotor].timeout=0;
				Timeouts[CurrentMotor] = 0;
			}
			break;
		}

		case 15:
		{
/* Wait, til CurrentMotor moves or timeout (maybe the CurrentMotor is already in endposition!)*/
			if(   (Motors[CurrentMotor].Moving == TRUE)
			   && (Motors[CurrentMotor].Error  == FALSE) )
			{
				Motors[CurrentMotor].ReferenceStep = 16;
				Motors[CurrentMotor].timeout = 0;
				break;
			}
			Motors[CurrentMotor].timeout++;
/* no movement after 12*cyclic time*/
			if(Motors[CurrentMotor].timeout >= TIMEOUT)
			{
				Motors[CurrentMotor].ReferenceStep = 16;
				Motors[CurrentMotor].timeout = 0;
			}
			break;
		}
		case 16:
		{
/* Wait, till CurrentMotor is stopped by obstacle */
/*
 * paperremove vertical: wait for sensor "up"
 */
			if( GlobalParameter.EnablePaletteLoading && (CurrentMotor == PAPERREMOVE_VERTICAL))
			{
				if(In_PaperRemoveUp)
				{
					Motors[CurrentMotor].ReferenceStep = 20;
					Timeouts[CurrentMotor] = 0;
					break;
				}
				Timeouts[CurrentMotor]++;
/* check for timeout */
				if(Timeouts[CurrentMotor] >= 20000) /*20 s*/
				{
					Motors[CurrentMotor].ReferenceStep = 17;
					Timeouts[CurrentMotor] = 0;
					break;
				}
			}
			else
			{
				if((Motors[CurrentMotor].Moving == 0) && (Motors[CurrentMotor].Error == 0))
				{
					Motors[CurrentMotor].ReferenceStep=20;
					Timeouts[CurrentMotor] = 0;
				}
			}
			break;
		}
/* special: Errorhandling PAPERREMOVE_VERTICAL */
		case 17:
		{
			if( SendMotorCmd(CurrentMotor, CMD_STOP, FALSE, 0L) )
			{
				Motors[CurrentMotor].ReferenceStep = 0;
				Motors[CurrentMotor].StartRef = FALSE;
				ShowMessage(94,0,95,CAUTION,OKONLY,TRUE);
			}
			break;
		}
		case 20:
		{
			if( SendMotorCmd(CurrentMotor, CMD_HOME, FALSE, 0L) )
			{
				Motors[CurrentMotor].ReferenceStep = 21;
			}
			break;
		}
		case 21:
		{
			if( SendMotorCmd(CurrentMotor, CMD_STOP, FALSE, 0L) )
			{
				Motors[CurrentMotor].ReferenceStep = 22;
			}
			break;
		}
		case 22:
		{
/* Wait, till sending is ready and CurrentMotor doesn't move*/
			if(Motors[CurrentMotor].Moving == FALSE)
			{
				if( GlobalParameter.EnablePaletteLoading && (CurrentMotor == PAPERREMOVE_VERTICAL))
					Motors[CurrentMotor].ReferenceStep = 110;
				else
				if(CurrentMotor == ADJUSTER || CurrentMotor == CONVEYORBELT)
					Motors[CurrentMotor].ReferenceStep = 30;
				else
					Motors[CurrentMotor].ReferenceStep = 23;
			}
			break;
		}
/****************************************************************/
/* special steps for Paperremove vertical */
/****************************************************************/
		case 110:
		{
/* move down (free from up-sensor */
			if( SendMotorCmd(CurrentMotor, CMD_MOVE_AT, TRUE, labs(Motors[CurrentMotor].Parameter.ReferenceSpeed / 10) ) )
			{
				Motors[CurrentMotor].ReferenceStep = 115;
				Timeouts[CurrentMotor] = 0;
			}
			break;
		}
/* wait for up-sensor to become free */
/* TODO timeout handling */
		case 115:
		{
			if(!In_PaperRemoveUp)
			{
				Motors[CurrentMotor].ReferenceStep = 120;
				Timeouts[CurrentMotor] = 0;
				break;
			}
			break;
		}
/* set 0-Pos on the fly*/
		case 120:
		{
			if( SendMotorCmd(CurrentMotor, CMD_HOME, FALSE, 0L) )
			{
				Motors[CurrentMotor].ReferenceStep = 121;
			}
			break;
		}
		case 121:
		{
			if( SendMotorCmd(CurrentMotor, CMD_STOP, FALSE, 0L) )
			{
				Motors[CurrentMotor].ReferenceStep = 23;
			}
			break;
		}
/****************************************************************/
/****************************************************************/

		case 23:
		{
			DINT tmpval;
			if( GlobalParameter.EnablePaletteLoading && (CurrentMotor == PAPERREMOVE_VERTICAL))
				tmpval = 0 - labs(Motors[CurrentMotor].Parameter.ReferenceOffset);
			else
				tmpval = labs(Motors[CurrentMotor].Parameter.ReferenceOffset);

			if( SendMotorCmd(CurrentMotor, CMD_RELATIVE_POS, TRUE, tmpval) )
			{
				Motors[CurrentMotor].ReferenceStep = 24;
			}
			break;
		}
		case 24:
		{
			if( SendMotorCmd(CurrentMotor, CMD_START_MOTION, FALSE, 0L) )
			{
				Motors[CurrentMotor].timeout = 0;
				Motors[CurrentMotor].ReferenceStep = 25;
			}
			break;
		}
		case 25:
		{
/* Wait, till sending is ready and CurrentMotor doesn't move*/
			Motors[CurrentMotor].timeout++;
			if(Motors[CurrentMotor].timeout > WAITTIME )
			{
				Motors[CurrentMotor].ReferenceStep = 26;
			}
			break;
		}

		case 26:
		{
/* Wait, till sending is ready and CurrentMotor doesn't move*/
			if(SerialCmd.Send == FALSE && Motors[CurrentMotor].Moving == FALSE)
			{
				if( GlobalParameter.EnablePaletteLoading && (CurrentMotor == PAPERREMOVE_VERTICAL))
					Motors[CurrentMotor].ReferenceStep = 27;
				else
					Motors[CurrentMotor].ReferenceStep = 30;
			}
			break;
		}

/****************************************************************/
/* special for Paperremove vertical */

		case 27:
		{
			if( SendMotorCmd(CurrentMotor, CMD_HOME, FALSE, 0L) )
			{
				Motors[CurrentMotor].ReferenceStep = 30;
			}
			break;
		}
/****************************************************************/

		case 30:
		{
			Motors[CurrentMotor].Parameter.Priority = OldPriority[CurrentMotor];
			Motors[CurrentMotor].Parameter.PositionWindow = OldPositionWindow[CurrentMotor];

			if( SendMotorCmd(CurrentMotor, CMD_PROPFACT, TRUE, Motors[CurrentMotor].Parameter.DefaultPropFact) )
			{
				Motors[CurrentMotor].ReferenceStep = 31;
			}
			break;
		}
		case 31:
		{
			if( SendMotorCmd(CurrentMotor, CMD_PEAK_CURRENT, TRUE, Motors[CurrentMotor].Parameter.DefaultPeekCurrent) )
			{
				Motors[CurrentMotor].ReferenceStep = 32;
			}
			break;
		}
		case 32:
		{
			if( SendMotorCmd(CurrentMotor, CMD_CONT_CURRENT, TRUE, Motors[CurrentMotor].Parameter.DefaultContCurrent) )
			{
				Motors[CurrentMotor].ReferenceStep = 33;
			}
			break;
		}
		case 33:
		{
			if( SendMotorCmd(CurrentMotor, CMD_ACCELERATION, TRUE, Motors[CurrentMotor].Parameter.DefaultAcceleration) )
			{
				Motors[CurrentMotor].ReferenceStep = 34;
			}
			break;
		}
		case 34:
		{
			if( SendMotorCmd(CurrentMotor, CMD_SPEED, TRUE, Motors[CurrentMotor].Parameter.MaximumSpeed) )
			{
				Motors[CurrentMotor].ReferenceStep = 35;
			}
			break;
		}
		case 35:
		{
			Motors[CurrentMotor].ReferenceStep = 0;
			Motors[CurrentMotor].StartRef = FALSE;
			Motors[CurrentMotor].ReferenceOk = TRUE;
			break;
		}
	}

	CurrentMotor++;

	if(   (CurrentMotor == FEEDER_HORIZONTAL)
	   && (GlobalParameter.FlexibleFeeder == FALSE) )
		CurrentMotor++;

	if(CurrentMotor == SHUTTLE)
		CurrentMotor++;

	if(CurrentMotor == ADJUSTER)
		CurrentMotor++;

	if(   (CurrentMotor == DELOADER_TURN)
	   && (GlobalParameter.DeloaderTurnStation != DELOADER_AND_TURNSTATION) )
		CurrentMotor++;

	if(   (CurrentMotor == DELOADER_HORIZONTAL)
	   && (GlobalParameter.DeloaderTurnStation == NO_DELOADER) )
		CurrentMotor++;

	if(CurrentMotor > MotorsConnected)
		CurrentMotor = FEEDER_VERTICAL;

}
/****************************************************************************/
/**                                                                        **/
/**                                 EOF                                    **/
/**                                                                        **/
/****************************************************************************/
```
